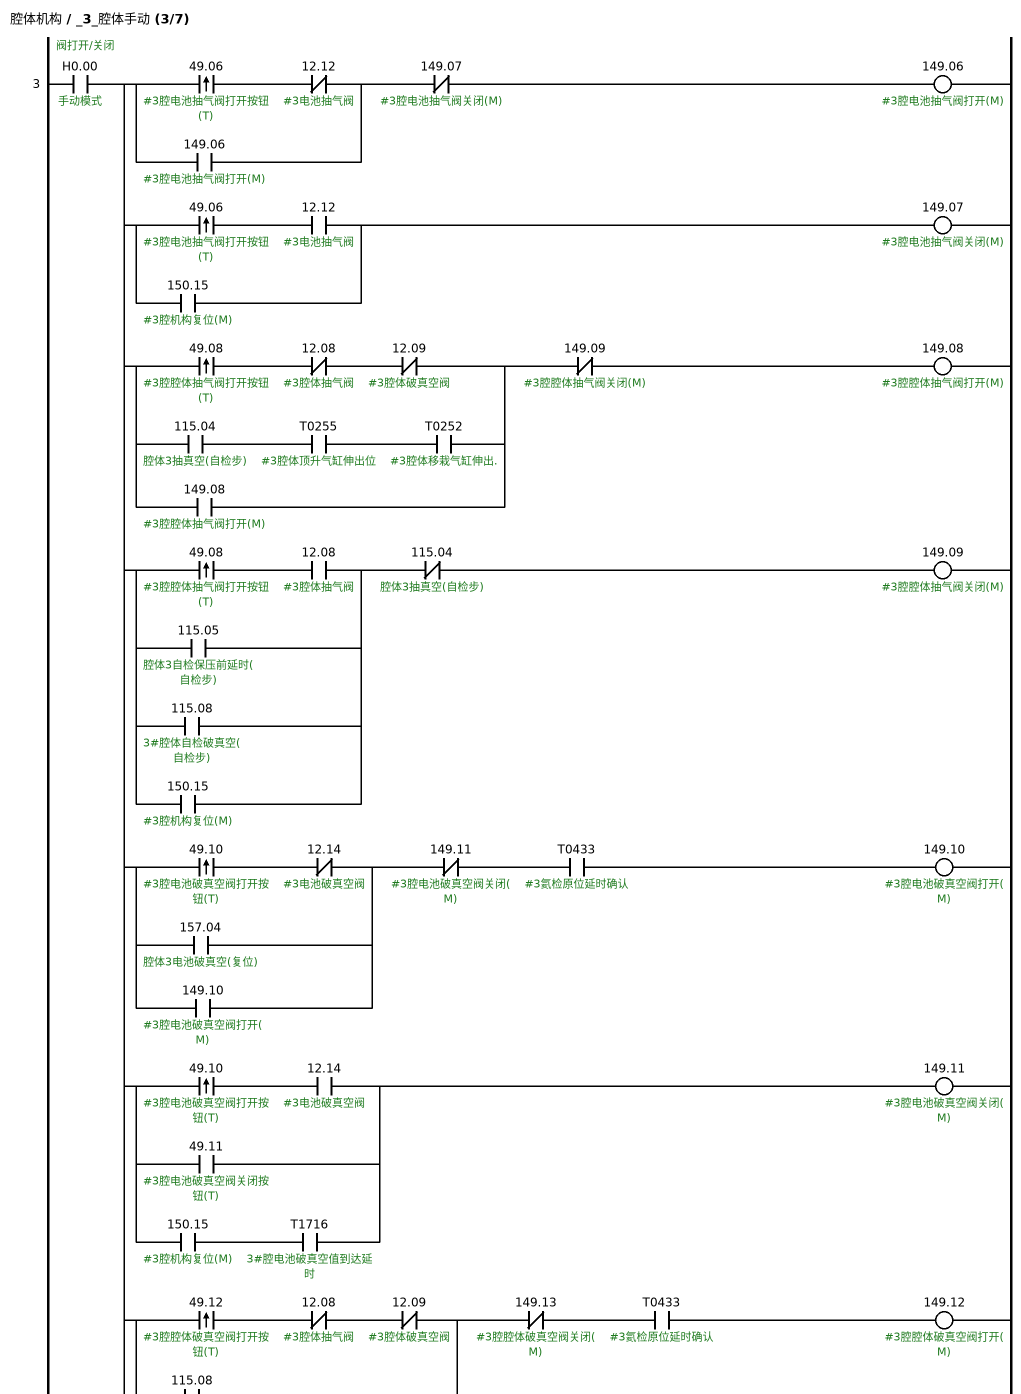
; [picture p264: 腔体机构 / _3_腔体手动, rungs 3-3]

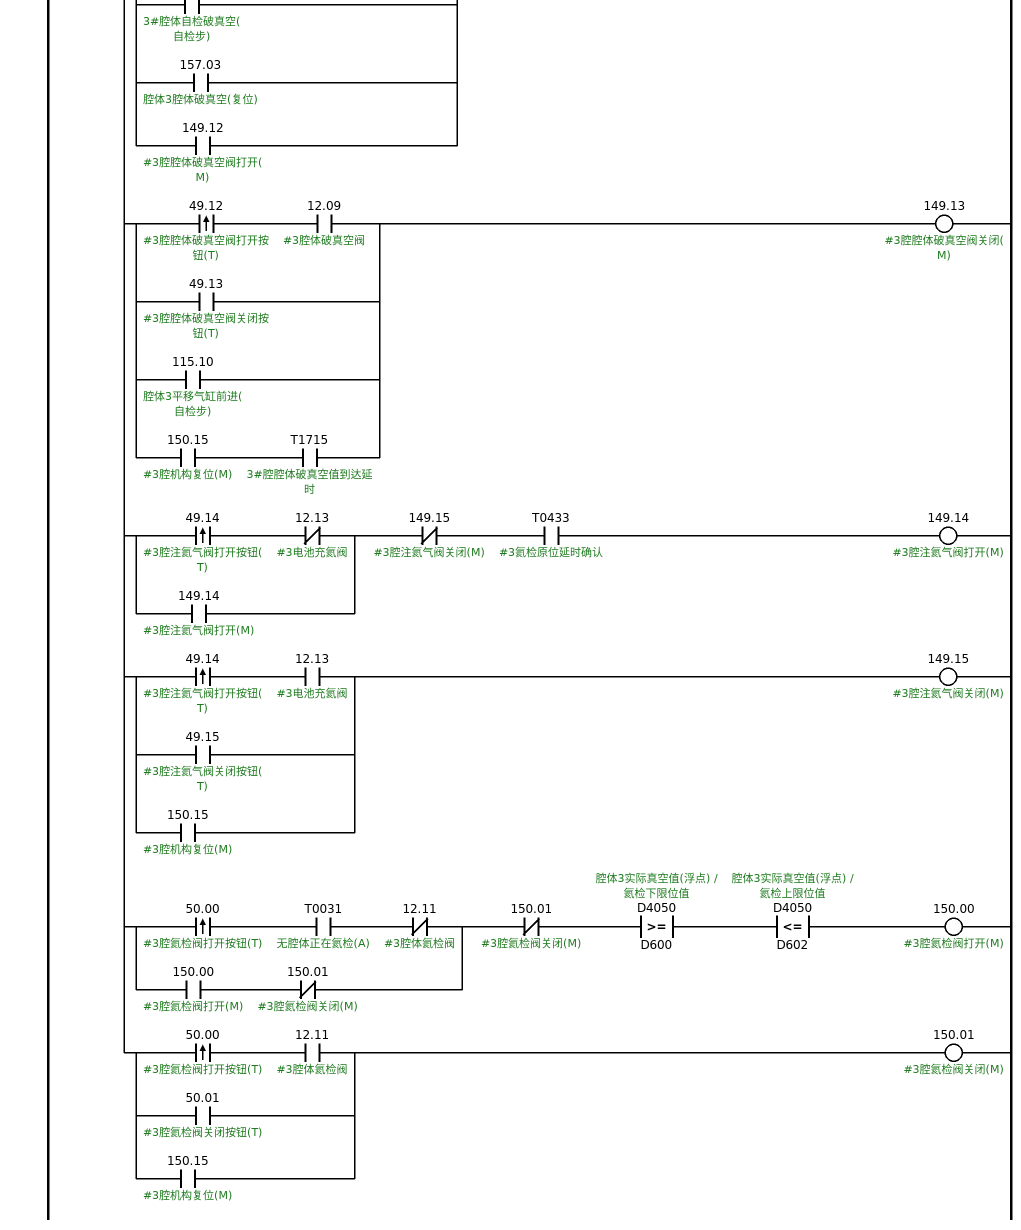
; rung 3: 阀打开/关闭
LD H0.00  ; 手动模式
OUT TR0
@LD 49.06  ; #3腔电池抽气阀打开按钮(T)
ANDNOT 12.12  ; #3电池抽气阀
OR 149.06  ; #3腔电池抽气阀打开(M)
ANDLD
ANDNOT 149.07  ; #3腔电池抽气阀关闭(M)
OUT 149.06  ; #3腔电池抽气阀打开(M)
LD TR0
@LD 49.06  ; #3腔电池抽气阀打开按钮(T)
AND 12.12  ; #3电池抽气阀
OR 150.15  ; #3腔机构复位(M)
ANDLD
OUT 149.07  ; #3腔电池抽气阀关闭(M)
LD TR0
@LD 49.08  ; #3腔腔体抽气阀打开按钮(T)
ANDNOT 12.08  ; #3腔体抽气阀
ANDNOT 12.09  ; #3腔体破真空阀
LD 115.04  ; 腔体3抽真空(自检步)
AND T0255  ; #3腔体顶升气缸伸出位
AND T0252  ; #3腔体移栽气缸伸出.
ORLD
OR 149.08  ; #3腔腔体抽气阀打开(M)
ANDLD
ANDNOT 149.09  ; #3腔腔体抽气阀关闭(M)
OUT 149.08  ; #3腔腔体抽气阀打开(M)
LD TR0
@LD 49.08  ; #3腔腔体抽气阀打开按钮(T)
AND 12.08  ; #3腔体抽气阀
OR 115.05  ; 腔体3自检保压前延时(自检步)
OR 115.08  ; 3#腔体自检破真空(自检步)
OR 150.15  ; #3腔机构复位(M)
ANDLD
ANDNOT 115.04  ; 腔体3抽真空(自检步)
OUT 149.09  ; #3腔腔体抽气阀关闭(M)
LD TR0
@LD 49.10  ; #3腔电池破真空阀打开按钮(T)
ANDNOT 12.14  ; #3电池破真空阀
OR 157.04  ; 腔体3电池破真空(复位)
OR 149.10  ; #3腔电池破真空阀打开(M)
ANDLD
ANDNOT 149.11  ; #3腔电池破真空阀关闭(M)
AND T0433  ; #3氦检原位延时确认
OUT 149.10  ; #3腔电池破真空阀打开(M)
LD TR0
@LD 49.10  ; #3腔电池破真空阀打开按钮(T)
AND 12.14  ; #3电池破真空阀
OR 49.11  ; #3腔电池破真空阀关闭按钮(T)
LD 150.15  ; #3腔机构复位(M)
AND T1716  ; 3#腔电池破真空值到达延时
ORLD
ANDLD
OUT 149.11  ; #3腔电池破真空阀关闭(M)
LD TR0
@LD 49.12  ; #3腔腔体破真空阀打开按钮(T)
ANDNOT 12.08  ; #3腔体抽气阀
ANDNOT 12.09  ; #3腔体破真空阀
OR 115.08  ; 3#腔体自检破真空(自检步)
OR 157.03  ; 腔体3腔体破真空(复位)
OR 149.12  ; #3腔腔体破真空阀打开(M)
ANDLD
ANDNOT 149.13  ; #3腔腔体破真空阀关闭(M)
AND T0433  ; #3氦检原位延时确认
OUT 149.12  ; #3腔腔体破真空阀打开(M)
LD TR0
@LD 49.12  ; #3腔腔体破真空阀打开按钮(T)
AND 12.09  ; #3腔体破真空阀
OR 49.13  ; #3腔腔体破真空阀关闭按钮(T)
OR 115.10  ; 腔体3平移气缸前进(自检步)
LD 150.15  ; #3腔机构复位(M)
AND T1715  ; 3#腔腔体破真空值到达延时
ORLD
ANDLD
OUT 149.13  ; #3腔腔体破真空阀关闭(M)
LD TR0
@LD 49.14  ; #3腔注氦气阀打开按钮(T)
ANDNOT 12.13  ; #3电池充氦阀
OR 149.14  ; #3腔注氦气阀打开(M)
ANDLD
ANDNOT 149.15  ; #3腔注氦气阀关闭(M)
AND T0433  ; #3氦检原位延时确认
OUT 149.14  ; #3腔注氦气阀打开(M)
LD TR0
@LD 49.14  ; #3腔注氦气阀打开按钮(T)
AND 12.13  ; #3电池充氦阀
OR 49.15  ; #3腔注氦气阀关闭按钮(T)
OR 150.15  ; #3腔机构复位(M)
ANDLD
OUT 149.15  ; #3腔注氦气阀关闭(M)
LD TR0
@LD 50.00  ; #3腔氦检阀打开按钮(T)
AND T0031  ; 无腔体正在氦检(A)
ANDNOT 12.11  ; #3腔体氦检阀
LD 150.00  ; #3腔氦检阀打开(M)
ANDNOT 150.01  ; #3腔氦检阀关闭(M)
ORLD
ANDLD
ANDNOT 150.01  ; #3腔氦检阀关闭(M)
AND>=F(334) D4050 D600  ; 腔体3实际真空值(浮点), 氦检下限位值
AND<=F(332) D4050 D602  ; 腔体3实际真空值(浮点), 氦检上限位值
OUT 150.00  ; #3腔氦检阀打开(M)
LD TR0
@LD 50.00  ; #3腔氦检阀打开按钮(T)
AND 12.11  ; #3腔体氦检阀
OR 50.01  ; #3腔氦检阀关闭按钮(T)
OR 150.15  ; #3腔机构复位(M)
ANDLD
OUT 150.01  ; #3腔氦检阀关闭(M)

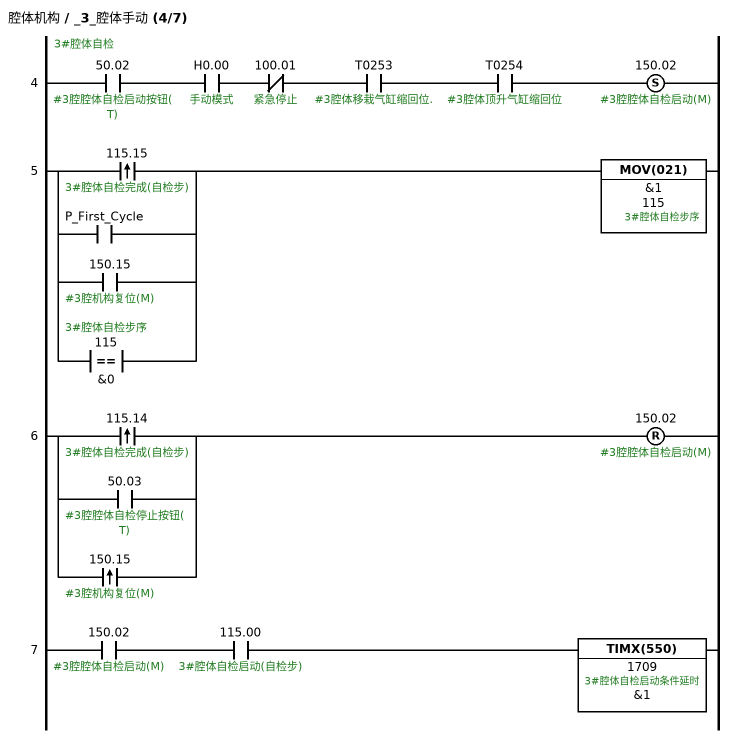
; rung 4: 3#腔体自检
LD 50.02  ; #3腔腔体自检启动按钮(T)
AND H0.00  ; 手动模式
ANDNOT 100.01  ; 紧急停止
AND T0253  ; #3腔体移栽气缸缩回位.
AND T0254  ; #3腔体顶升气缸缩回位
SET 150.02  ; #3腔腔体自检启动(M)
; rung 5
@LD 115.15  ; 3#腔体自检完成(自检步)
OR P_First_Cycle
OR 150.15  ; #3腔机构复位(M)
OR=(300) 115 &0  ; 3#腔体自检步序
MOV(021) &1 115  ; 3#腔体自检步序
; rung 6
@LD 115.14  ; 3#腔体自检完成(自检步)
OR 50.03  ; #3腔腔体自检停止按钮(T)
@OR 150.15  ; #3腔机构复位(M)
RSET 150.02  ; #3腔腔体自检启动(M)
; rung 7
LD 150.02  ; #3腔腔体自检启动(M)
AND 115.00  ; 3#腔体自检启动(自检步)
TIMX(550) 1709 &1  ; 3#腔体自检启动条件延时

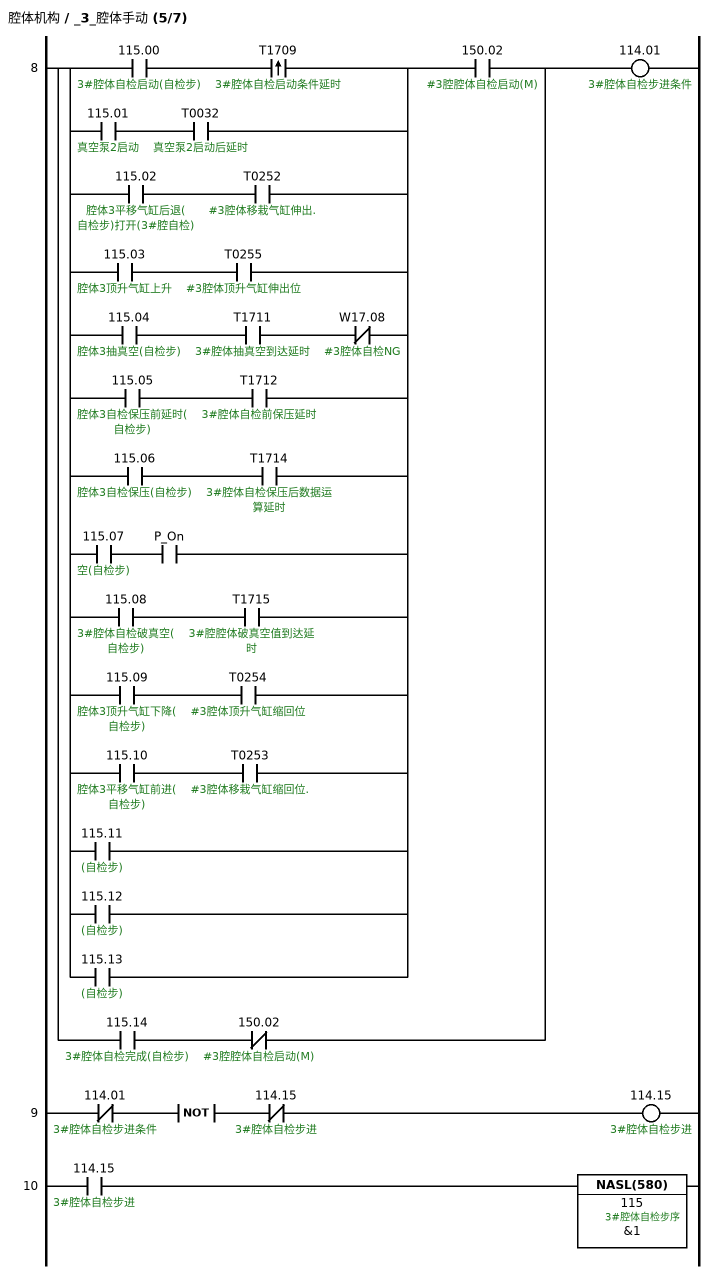
; rung 8
LD 115.00  ; 3#腔体自检启动(自检步)
@AND T1709  ; 3#腔体自检启动条件延时
LD 115.01  ; 真空泵2启动
AND T0032  ; 真空泵2启动后延时
ORLD
LD 115.02  ; 腔体3平移气缸后退(自检步)打开(3#腔自检)
AND T0252  ; #3腔体移栽气缸伸出.
ORLD
LD 115.03  ; 腔体3顶升气缸上升
AND T0255  ; #3腔体顶升气缸伸出位
ORLD
LD 115.04  ; 腔体3抽真空(自检步)
AND T1711  ; 3#腔体抽真空到达延时
ANDNOT W17.08  ; #3腔体自检NG
ORLD
LD 115.05  ; 腔体3自检保压前延时(自检步)
AND T1712  ; 3#腔体自检前保压延时
ORLD
LD 115.06  ; 腔体3自检保压(自检步)
AND T1714  ; 3#腔体自检保压后数据运算延时
ORLD
LD 115.07  ; 空(自检步)
AND P_On
ORLD
LD 115.08  ; 3#腔体自检破真空(自检步)
AND T1715  ; 3#腔腔体破真空值到达延时
ORLD
LD 115.09  ; 腔体3顶升气缸下降(自检步)
AND T0254  ; #3腔体顶升气缸缩回位
ORLD
LD 115.10  ; 腔体3平移气缸前进(自检步)
AND T0253  ; #3腔体移栽气缸缩回位.
ORLD
OR 115.11  ; (自检步)
OR 115.12  ; (自检步)
OR 115.13  ; (自检步)
AND 150.02  ; #3腔腔体自检启动(M)
LD 115.14  ; 3#腔体自检完成(自检步)
ANDNOT 150.02  ; #3腔腔体自检启动(M)
ORLD
OUT 114.01  ; 3#腔体自检步进条件
; rung 9
LDNOT 114.01  ; 3#腔体自检步进条件
NOT(520)
ANDNOT 114.15  ; 3#腔体自检步进
OUT 114.15  ; 3#腔体自检步进
; rung 10
LD 114.15  ; 3#腔体自检步进
NASL(580) 115 &1  ; 3#腔体自检步序

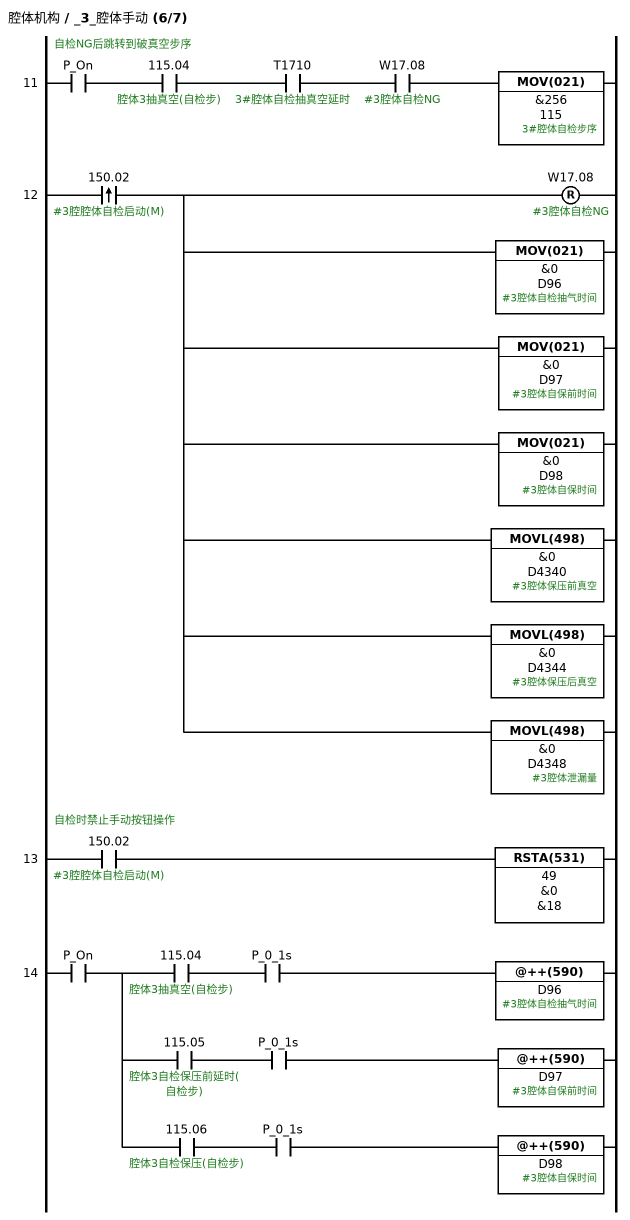
; rung 11: 自检NG后跳转到破真空步序
LD P_On
AND 115.04  ; 腔体3抽真空(自检步)
AND T1710  ; 3#腔体自检抽真空延时
AND W17.08  ; #3腔体自检NG
MOV(021) &256 115  ; 3#腔体自检步序
; rung 12
@LD 150.02  ; #3腔腔体自检启动(M)
RSET W17.08  ; #3腔体自检NG
MOV(021) &0 D96  ; #3腔体自检抽气时间
MOV(021) &0 D97  ; #3腔体自保前时间
MOV(021) &0 D98  ; #3腔体自保时间
MOVL(498) &0 D4340  ; #3腔体保压前真空
MOVL(498) &0 D4344  ; #3腔体保压后真空
MOVL(498) &0 D4348  ; #3腔体泄漏量
; rung 13: 自检时禁止手动按钮操作
LD 150.02  ; #3腔腔体自检启动(M)
RSTA(531) 49 &0 &18
; rung 14
LD P_On
OUT TR0
AND 115.04  ; 腔体3抽真空(自检步)
AND P_0_1s
@++(590) D96  ; #3腔体自检抽气时间
LD TR0
AND 115.05  ; 腔体3自检保压前延时(自检步)
AND P_0_1s
@++(590) D97  ; #3腔体自保前时间
LD TR0
AND 115.06  ; 腔体3自检保压(自检步)
AND P_0_1s
@++(590) D98  ; #3腔体自保时间

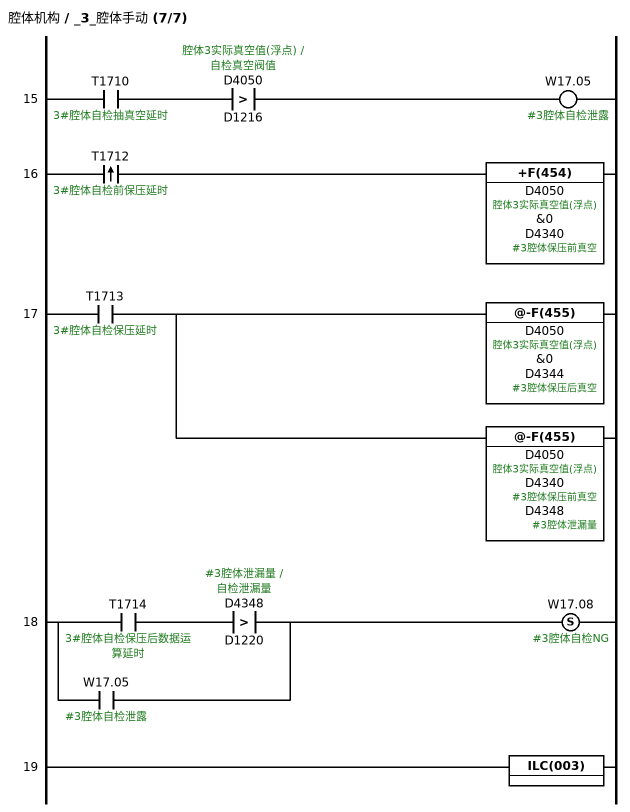
; rung 15
LD T1710  ; 3#腔体自检抽真空延时
AND>F(333) D4050 D1216  ; 腔体3实际真空值(浮点), 自检真空阀值
OUT W17.05  ; #3腔体自检泄露
; rung 16
@LD T1712  ; 3#腔体自检前保压延时
+F(454) D4050 &0 D4340  ; 腔体3实际真空值(浮点), #3腔体保压前真空
; rung 17
LD T1713  ; 3#腔体自检保压延时
@-F(455) D4050 &0 D4344  ; 腔体3实际真空值(浮点), #3腔体保压后真空
@-F(455) D4050 D4340 D4348  ; 腔体3实际真空值(浮点), #3腔体保压前真空, #3腔体泄漏量
; rung 18
LD T1714  ; 3#腔体自检保压后数据运算延时
AND>F(333) D4348 D1220  ; #3腔体泄漏量, 自检泄漏量
OR W17.05  ; #3腔体自检泄露
SET W17.08  ; #3腔体自检NG
; rung 19
ILC(003)

### Section _4_腔体手动

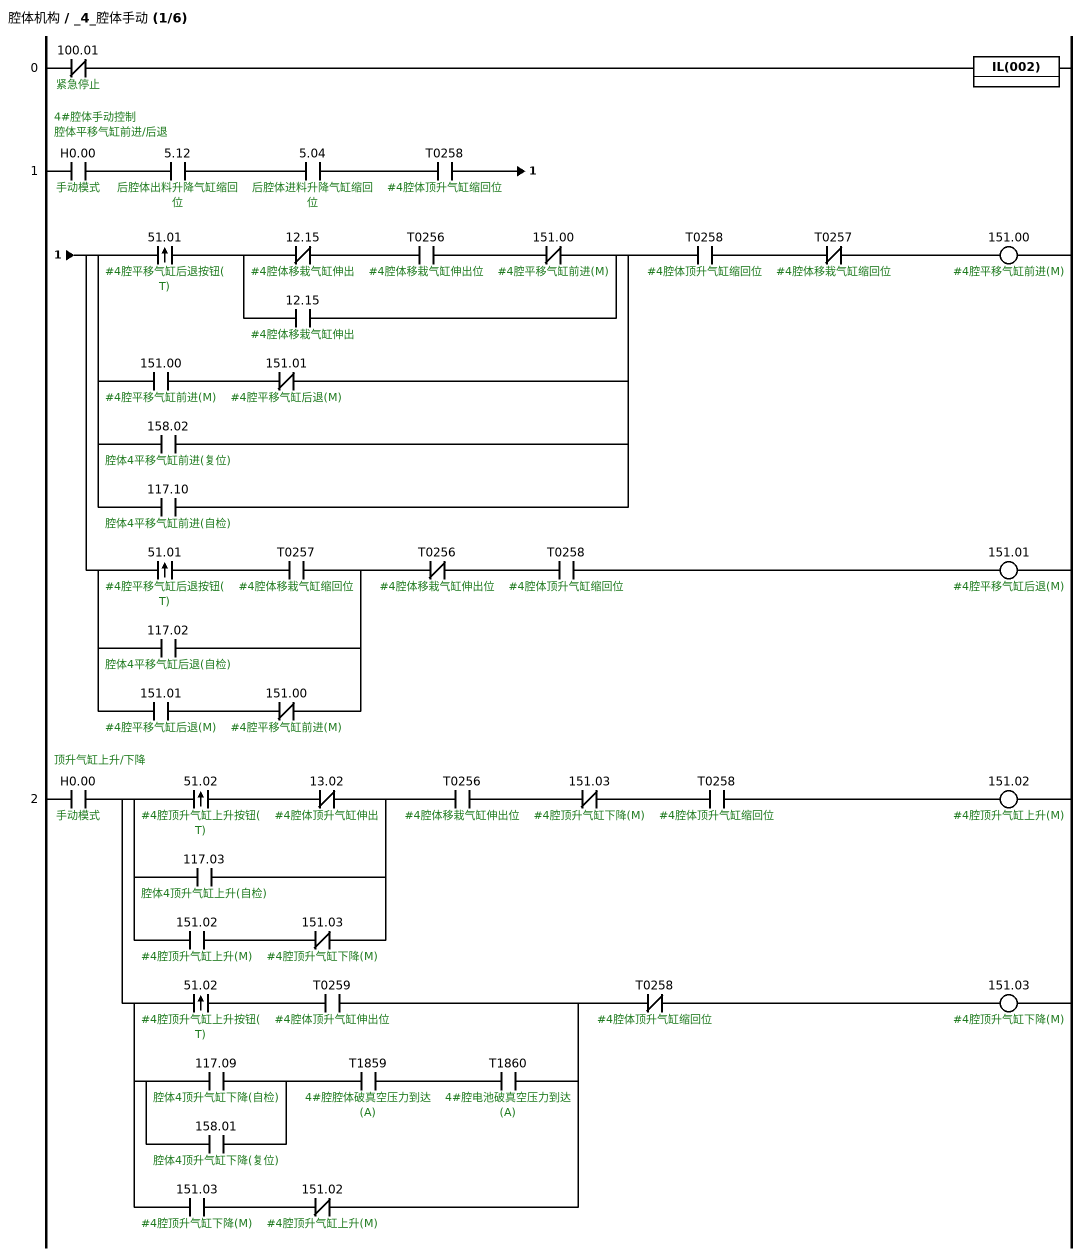
; rung 0
LDNOT 100.01  ; 紧急停止
IL(002)
; rung 1: 4#腔体手动控制 / 腔体平移气缸前进/后退
LD H0.00  ; 手动模式
AND 5.12  ; 后腔体出料升降气缸缩回位
AND 5.04  ; 后腔体进料升降气缸缩回位
AND T0258  ; #4腔体顶升气缸缩回位
OUT TR0
@LD 51.01  ; #4腔平移气缸后退按钮(T)
LDNOT 12.15  ; #4腔体移栽气缸伸出
AND T0256  ; #4腔体移栽气缸伸出位
ANDNOT 151.00  ; #4腔平移气缸前进(M)
OR 12.15  ; #4腔体移栽气缸伸出
ANDLD
LD 151.00  ; #4腔平移气缸前进(M)
ANDNOT 151.01  ; #4腔平移气缸后退(M)
ORLD
OR 158.02  ; 腔体4平移气缸前进(复位)
OR 117.10  ; 腔体4平移气缸前进(自检)
ANDLD
AND T0258  ; #4腔体顶升气缸缩回位
ANDNOT T0257  ; #4腔体移栽气缸缩回位
OUT 151.00  ; #4腔平移气缸前进(M)
LD TR0
@LD 51.01  ; #4腔平移气缸后退按钮(T)
AND T0257  ; #4腔体移栽气缸缩回位
OR 117.02  ; 腔体4平移气缸后退(自检)
LD 151.01  ; #4腔平移气缸后退(M)
ANDNOT 151.00  ; #4腔平移气缸前进(M)
ORLD
ANDLD
ANDNOT T0256  ; #4腔体移栽气缸伸出位
AND T0258  ; #4腔体顶升气缸缩回位
OUT 151.01  ; #4腔平移气缸后退(M)
; rung 2: 顶升气缸上升/下降
LD H0.00  ; 手动模式
OUT TR0
@LD 51.02  ; #4腔顶升气缸上升按钮(T)
ANDNOT 13.02  ; #4腔体顶升气缸伸出
OR 117.03  ; 腔体4顶升气缸上升(自检)
LD 151.02  ; #4腔顶升气缸上升(M)
ANDNOT 151.03  ; #4腔顶升气缸下降(M)
ORLD
ANDLD
AND T0256  ; #4腔体移栽气缸伸出位
ANDNOT 151.03  ; #4腔顶升气缸下降(M)
AND T0258  ; #4腔体顶升气缸缩回位
OUT 151.02  ; #4腔顶升气缸上升(M)
LD TR0
@LD 51.02  ; #4腔顶升气缸上升按钮(T)
AND T0259  ; #4腔体顶升气缸伸出位
LD 117.09  ; 腔体4顶升气缸下降(自检)
OR 158.01  ; 腔体4顶升气缸下降(复位)
AND T1859  ; 4#腔腔体破真空压力到达(A)
AND T1860  ; 4#腔电池破真空压力到达(A)
ORLD
LD 151.03  ; #4腔顶升气缸下降(M)
ANDNOT 151.02  ; #4腔顶升气缸上升(M)
ORLD
ANDLD
ANDNOT T0258  ; #4腔体顶升气缸缩回位
OUT 151.03  ; #4腔顶升气缸下降(M)

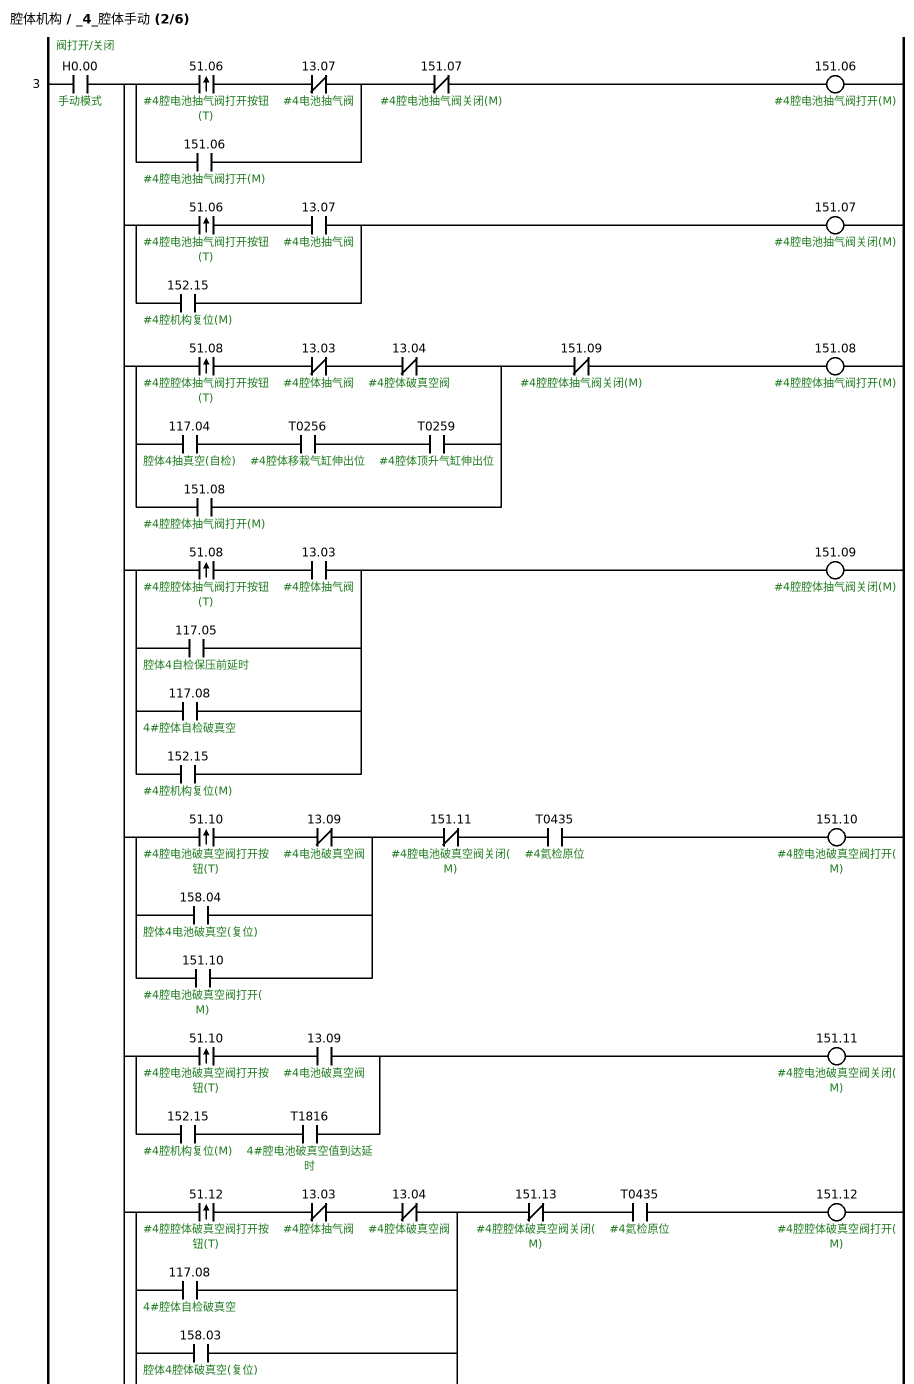

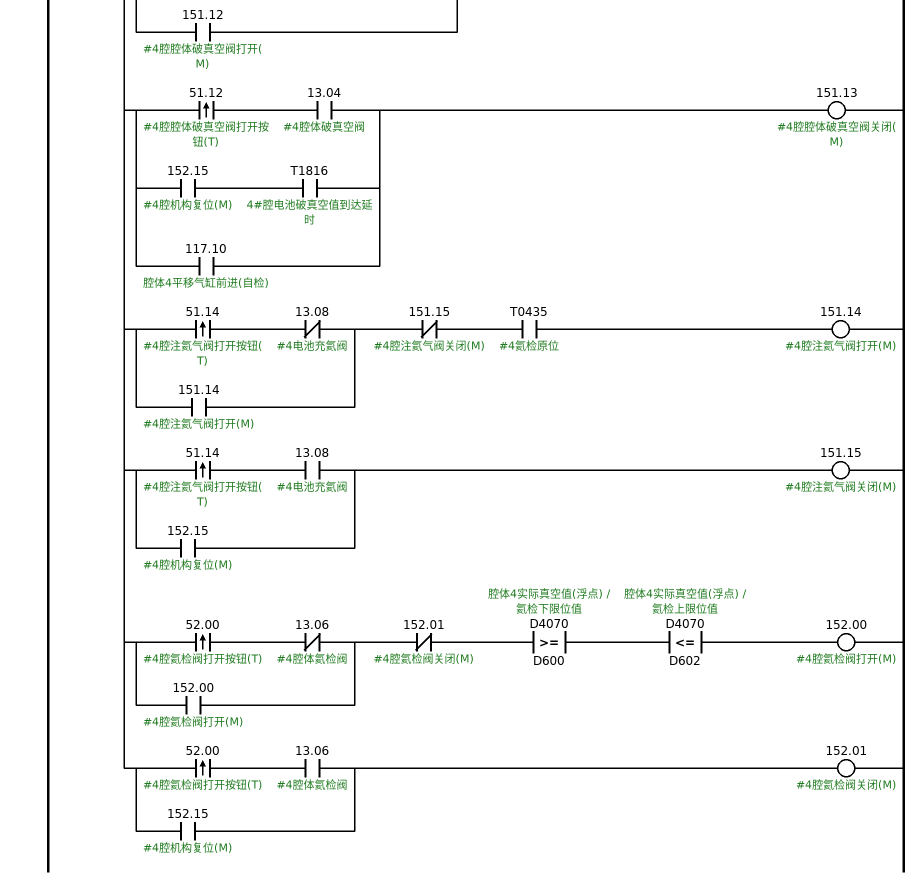
; rung 3: 阀打开/关闭
LD H0.00  ; 手动模式
OUT TR0
@LD 51.06  ; #4腔电池抽气阀打开按钮(T)
ANDNOT 13.07  ; #4电池抽气阀
OR 151.06  ; #4腔电池抽气阀打开(M)
ANDLD
ANDNOT 151.07  ; #4腔电池抽气阀关闭(M)
OUT 151.06  ; #4腔电池抽气阀打开(M)
LD TR0
@LD 51.06  ; #4腔电池抽气阀打开按钮(T)
AND 13.07  ; #4电池抽气阀
OR 152.15  ; #4腔机构复位(M)
ANDLD
OUT 151.07  ; #4腔电池抽气阀关闭(M)
LD TR0
@LD 51.08  ; #4腔腔体抽气阀打开按钮(T)
ANDNOT 13.03  ; #4腔体抽气阀
ANDNOT 13.04  ; #4腔体破真空阀
LD 117.04  ; 腔体4抽真空(自检)
AND T0256  ; #4腔体移栽气缸伸出位
AND T0259  ; #4腔体顶升气缸伸出位
ORLD
OR 151.08  ; #4腔腔体抽气阀打开(M)
ANDLD
ANDNOT 151.09  ; #4腔腔体抽气阀关闭(M)
OUT 151.08  ; #4腔腔体抽气阀打开(M)
LD TR0
@LD 51.08  ; #4腔腔体抽气阀打开按钮(T)
AND 13.03  ; #4腔体抽气阀
OR 117.05  ; 腔体4自检保压前延时
OR 117.08  ; 4#腔体自检破真空
OR 152.15  ; #4腔机构复位(M)
ANDLD
OUT 151.09  ; #4腔腔体抽气阀关闭(M)
LD TR0
@LD 51.10  ; #4腔电池破真空阀打开按钮(T)
ANDNOT 13.09  ; #4电池破真空阀
OR 158.04  ; 腔体4电池破真空(复位)
OR 151.10  ; #4腔电池破真空阀打开(M)
ANDLD
ANDNOT 151.11  ; #4腔电池破真空阀关闭(M)
AND T0435  ; #4氦检原位
OUT 151.10  ; #4腔电池破真空阀打开(M)
LD TR0
@LD 51.10  ; #4腔电池破真空阀打开按钮(T)
AND 13.09  ; #4电池破真空阀
LD 152.15  ; #4腔机构复位(M)
AND T1816  ; 4#腔电池破真空值到达延时
ORLD
ANDLD
OUT 151.11  ; #4腔电池破真空阀关闭(M)
LD TR0
@LD 51.12  ; #4腔腔体破真空阀打开按钮(T)
ANDNOT 13.03  ; #4腔体抽气阀
ANDNOT 13.04  ; #4腔体破真空阀
OR 117.08  ; 4#腔体自检破真空
OR 158.03  ; 腔体4腔体破真空(复位)
OR 151.12  ; #4腔腔体破真空阀打开(M)
ANDLD
ANDNOT 151.13  ; #4腔腔体破真空阀关闭(M)
AND T0435  ; #4氦检原位
OUT 151.12  ; #4腔腔体破真空阀打开(M)
LD TR0
@LD 51.12  ; #4腔腔体破真空阀打开按钮(T)
AND 13.04  ; #4腔体破真空阀
LD 152.15  ; #4腔机构复位(M)
AND T1816  ; 4#腔电池破真空值到达延时
ORLD
OR 117.10  ; 腔体4平移气缸前进(自检)
ANDLD
OUT 151.13  ; #4腔腔体破真空阀关闭(M)
LD TR0
@LD 51.14  ; #4腔注氦气阀打开按钮(T)
ANDNOT 13.08  ; #4电池充氦阀
OR 151.14  ; #4腔注氦气阀打开(M)
ANDLD
ANDNOT 151.15  ; #4腔注氦气阀关闭(M)
AND T0435  ; #4氦检原位
OUT 151.14  ; #4腔注氦气阀打开(M)
LD TR0
@LD 51.14  ; #4腔注氦气阀打开按钮(T)
AND 13.08  ; #4电池充氦阀
OR 152.15  ; #4腔机构复位(M)
ANDLD
OUT 151.15  ; #4腔注氦气阀关闭(M)
LD TR0
@LD 52.00  ; #4腔氦检阀打开按钮(T)
ANDNOT 13.06  ; #4腔体氦检阀
OR 152.00  ; #4腔氦检阀打开(M)
ANDLD
ANDNOT 152.01  ; #4腔氦检阀关闭(M)
AND>=F(334) D4070 D600  ; 腔体4实际真空值(浮点), 氦检下限位值
AND<=F(332) D4070 D602  ; 腔体4实际真空值(浮点), 氦检上限位值
OUT 152.00  ; #4腔氦检阀打开(M)
LD TR0
@LD 52.00  ; #4腔氦检阀打开按钮(T)
AND 13.06  ; #4腔体氦检阀
OR 152.15  ; #4腔机构复位(M)
ANDLD
OUT 152.01  ; #4腔氦检阀关闭(M)

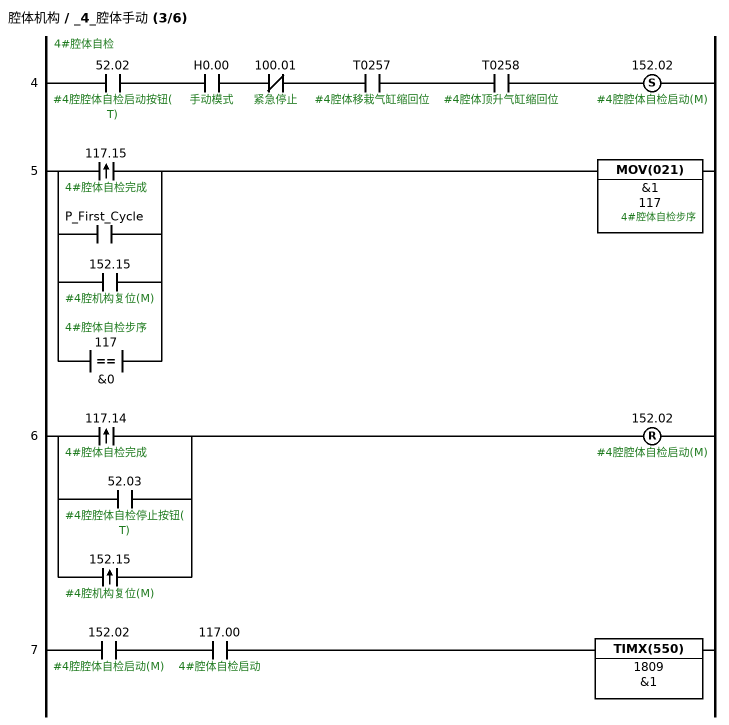
; rung 4: 4#腔体自检
LD 52.02  ; #4腔腔体自检启动按钮(T)
AND H0.00  ; 手动模式
ANDNOT 100.01  ; 紧急停止
AND T0257  ; #4腔体移栽气缸缩回位
AND T0258  ; #4腔体顶升气缸缩回位
SET 152.02  ; #4腔腔体自检启动(M)
; rung 5
@LD 117.15  ; 4#腔体自检完成
OR P_First_Cycle
OR 152.15  ; #4腔机构复位(M)
OR=(300) 117 &0  ; 4#腔体自检步序
MOV(021) &1 117  ; 4#腔体自检步序
; rung 6
@LD 117.14  ; 4#腔体自检完成
OR 52.03  ; #4腔腔体自检停止按钮(T)
@OR 152.15  ; #4腔机构复位(M)
RSET 152.02  ; #4腔腔体自检启动(M)
; rung 7
LD 152.02  ; #4腔腔体自检启动(M)
AND 117.00  ; 4#腔体自检启动
TIMX(550) 1809 &1

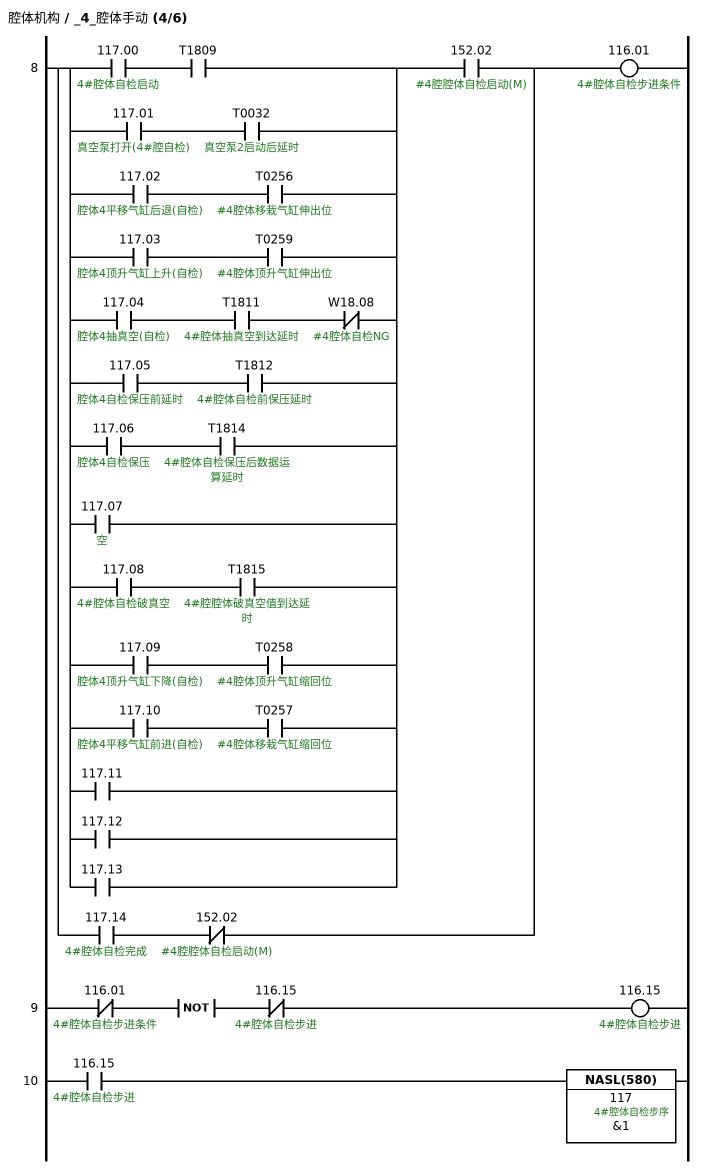
; rung 8
LD 117.00  ; 4#腔体自检启动
AND T1809
LD 117.01  ; 真空泵打开(4#腔自检)
AND T0032  ; 真空泵2启动后延时
ORLD
LD 117.02  ; 腔体4平移气缸后退(自检)
AND T0256  ; #4腔体移栽气缸伸出位
ORLD
LD 117.03  ; 腔体4顶升气缸上升(自检)
AND T0259  ; #4腔体顶升气缸伸出位
ORLD
LD 117.04  ; 腔体4抽真空(自检)
AND T1811  ; 4#腔体抽真空到达延时
ANDNOT W18.08  ; #4腔体自检NG
ORLD
LD 117.05  ; 腔体4自检保压前延时
AND T1812  ; 4#腔体自检前保压延时
ORLD
LD 117.06  ; 腔体4自检保压
AND T1814  ; 4#腔体自检保压后数据运算延时
ORLD
OR 117.07  ; 空
LD 117.08  ; 4#腔体自检破真空
AND T1815  ; 4#腔腔体破真空值到达延时
ORLD
LD 117.09  ; 腔体4顶升气缸下降(自检)
AND T0258  ; #4腔体顶升气缸缩回位
ORLD
LD 117.10  ; 腔体4平移气缸前进(自检)
AND T0257  ; #4腔体移栽气缸缩回位
ORLD
OR 117.11
OR 117.12
OR 117.13
AND 152.02  ; #4腔腔体自检启动(M)
LD 117.14  ; 4#腔体自检完成
ANDNOT 152.02  ; #4腔腔体自检启动(M)
ORLD
OUT 116.01  ; 4#腔体自检步进条件
; rung 9
LDNOT 116.01  ; 4#腔体自检步进条件
NOT(520)
ANDNOT 116.15  ; 4#腔体自检步进
OUT 116.15  ; 4#腔体自检步进
; rung 10
LD 116.15  ; 4#腔体自检步进
NASL(580) 117 &1  ; 4#腔体自检步序

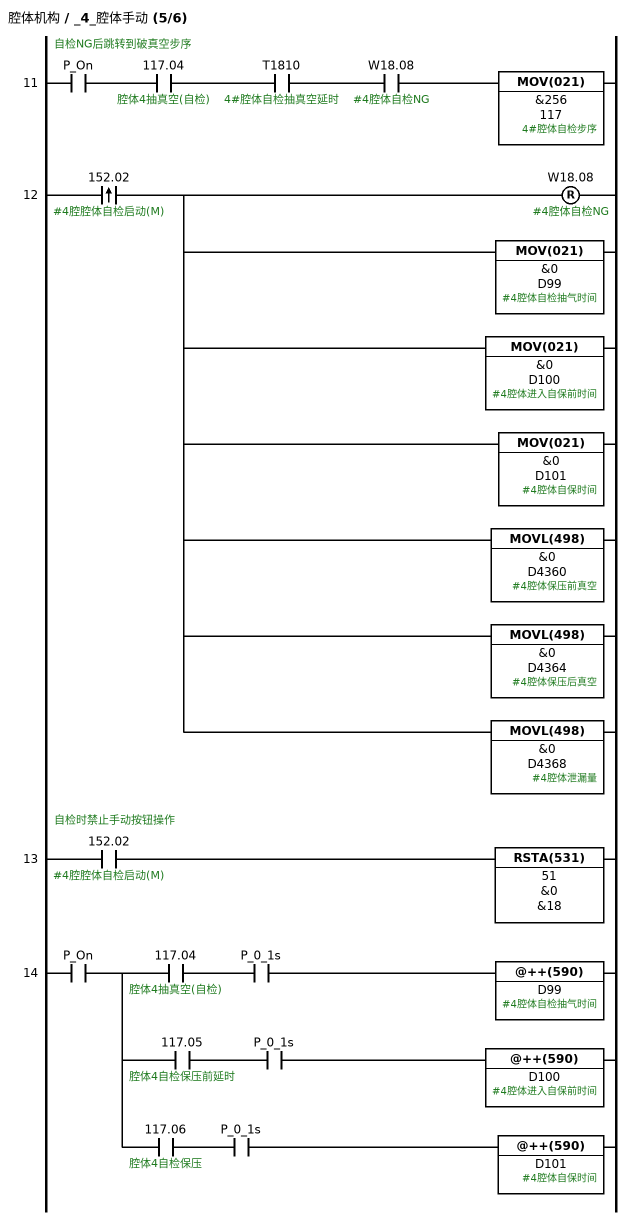
; rung 11: 自检NG后跳转到破真空步序
LD P_On
AND 117.04  ; 腔体4抽真空(自检)
AND T1810  ; 4#腔体自检抽真空延时
AND W18.08  ; #4腔体自检NG
MOV(021) &256 117  ; 4#腔体自检步序
; rung 12
@LD 152.02  ; #4腔腔体自检启动(M)
RSET W18.08  ; #4腔体自检NG
MOV(021) &0 D99  ; #4腔体自检抽气时间
MOV(021) &0 D100  ; #4腔体进入自保前时间
MOV(021) &0 D101  ; #4腔体自保时间
MOVL(498) &0 D4360  ; #4腔体保压前真空
MOVL(498) &0 D4364  ; #4腔体保压后真空
MOVL(498) &0 D4368  ; #4腔体泄漏量
; rung 13: 自检时禁止手动按钮操作
LD 152.02  ; #4腔腔体自检启动(M)
RSTA(531) 51 &0 &18
; rung 14
LD P_On
OUT TR0
AND 117.04  ; 腔体4抽真空(自检)
AND P_0_1s
@++(590) D99  ; #4腔体自检抽气时间
LD TR0
AND 117.05  ; 腔体4自检保压前延时
AND P_0_1s
@++(590) D100  ; #4腔体进入自保前时间
LD TR0
AND 117.06  ; 腔体4自检保压
AND P_0_1s
@++(590) D101  ; #4腔体自保时间

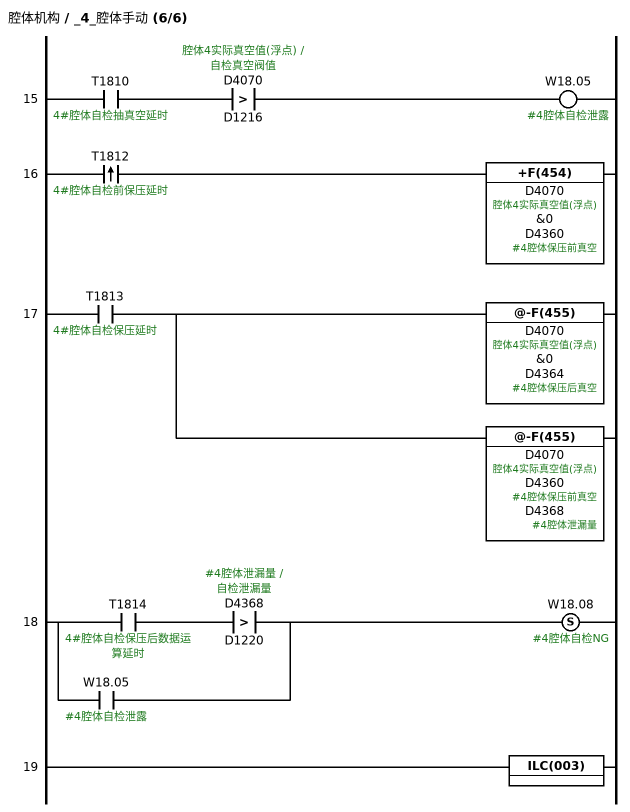
; rung 15
LD T1810  ; 4#腔体自检抽真空延时
AND>F(333) D4070 D1216  ; 腔体4实际真空值(浮点), 自检真空阀值
OUT W18.05  ; #4腔体自检泄露
; rung 16
@LD T1812  ; 4#腔体自检前保压延时
+F(454) D4070 &0 D4360  ; 腔体4实际真空值(浮点), #4腔体保压前真空
; rung 17
LD T1813  ; 4#腔体自检保压延时
@-F(455) D4070 &0 D4364  ; 腔体4实际真空值(浮点), #4腔体保压后真空
@-F(455) D4070 D4360 D4368  ; 腔体4实际真空值(浮点), #4腔体保压前真空, #4腔体泄漏量
; rung 18
LD T1814  ; 4#腔体自检保压后数据运算延时
AND>F(333) D4368 D1220  ; #4腔体泄漏量, 自检泄漏量
OR W18.05  ; #4腔体自检泄露
SET W18.08  ; #4腔体自检NG
; rung 19
ILC(003)

### Section _1_腔体自动

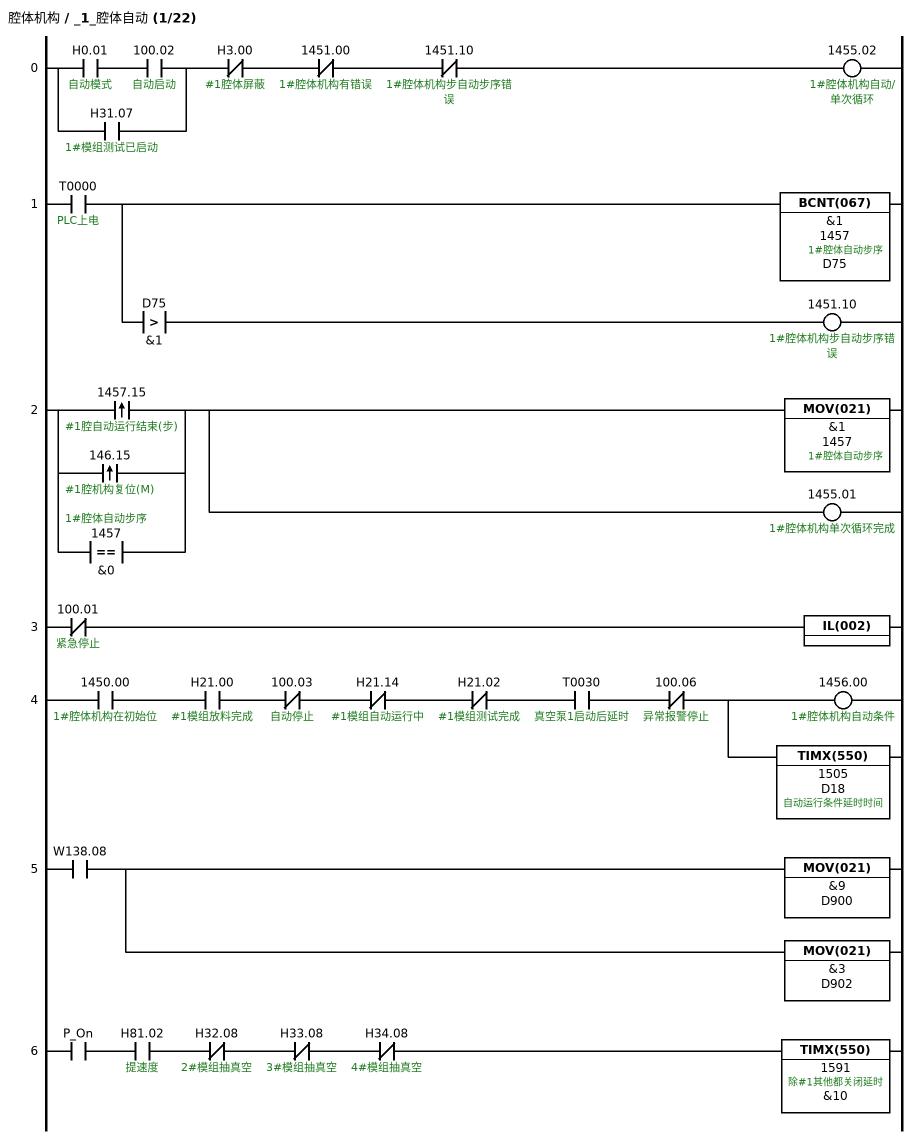
; rung 0
LD H0.01  ; 自动模式
AND 100.02  ; 自动启动
OR H31.07  ; 1#模组测试已启动
ANDNOT H3.00  ; #1腔体屏蔽
ANDNOT 1451.00  ; 1#腔体机构有错误
ANDNOT 1451.10  ; 1#腔体机构步自动步序错误
OUT 1455.02  ; 1#腔体机构自动/单次循环
; rung 1
LD T0000  ; PLC上电
BCNT(067) &1 1457 D75  ; 1#腔体自动步序
AND>(320) D75 &1
OUT 1451.10  ; 1#腔体机构步自动步序错误
; rung 2
@LD 1457.15  ; #1腔自动运行结束(步)
@OR 146.15  ; #1腔机构复位(M)
OR=(300) 1457 &0  ; 1#腔体自动步序
MOV(021) &1 1457  ; 1#腔体自动步序
OUT 1455.01  ; 1#腔体机构单次循环完成
; rung 3
LDNOT 100.01  ; 紧急停止
IL(002)
; rung 4
LD 1450.00  ; 1#腔体机构在初始位
AND H21.00  ; #1模组放料完成
ANDNOT 100.03  ; 自动停止
ANDNOT H21.14  ; #1模组自动运行中
ANDNOT H21.02  ; #1模组测试完成
AND T0030  ; 真空泵1启动后延时
ANDNOT 100.06  ; 异常报警停止
OUT 1456.00  ; 1#腔体机构自动条件
TIMX(550) 1505 D18  ; 自动运行条件延时时间
; rung 5
LD W138.08
MOV(021) &9 D900
MOV(021) &3 D902
; rung 6
LD P_On
AND H81.02  ; 提速度
ANDNOT H32.08  ; 2#模组抽真空
ANDNOT H33.08  ; 3#模组抽真空
ANDNOT H34.08  ; 4#模组抽真空
TIMX(550) 1591 &10  ; 除#1其他都关闭延时

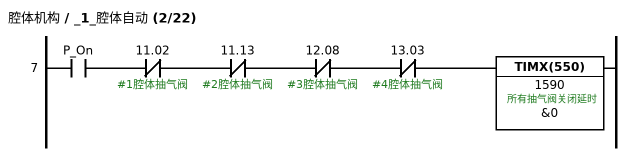
; rung 7
LD P_On
ANDNOT 11.02  ; #1腔体抽气阀
ANDNOT 11.13  ; #2腔体抽气阀
ANDNOT 12.08  ; #3腔体抽气阀
ANDNOT 13.03  ; #4腔体抽气阀
TIMX(550) 1590 &0  ; 所有抽气阀关闭延时

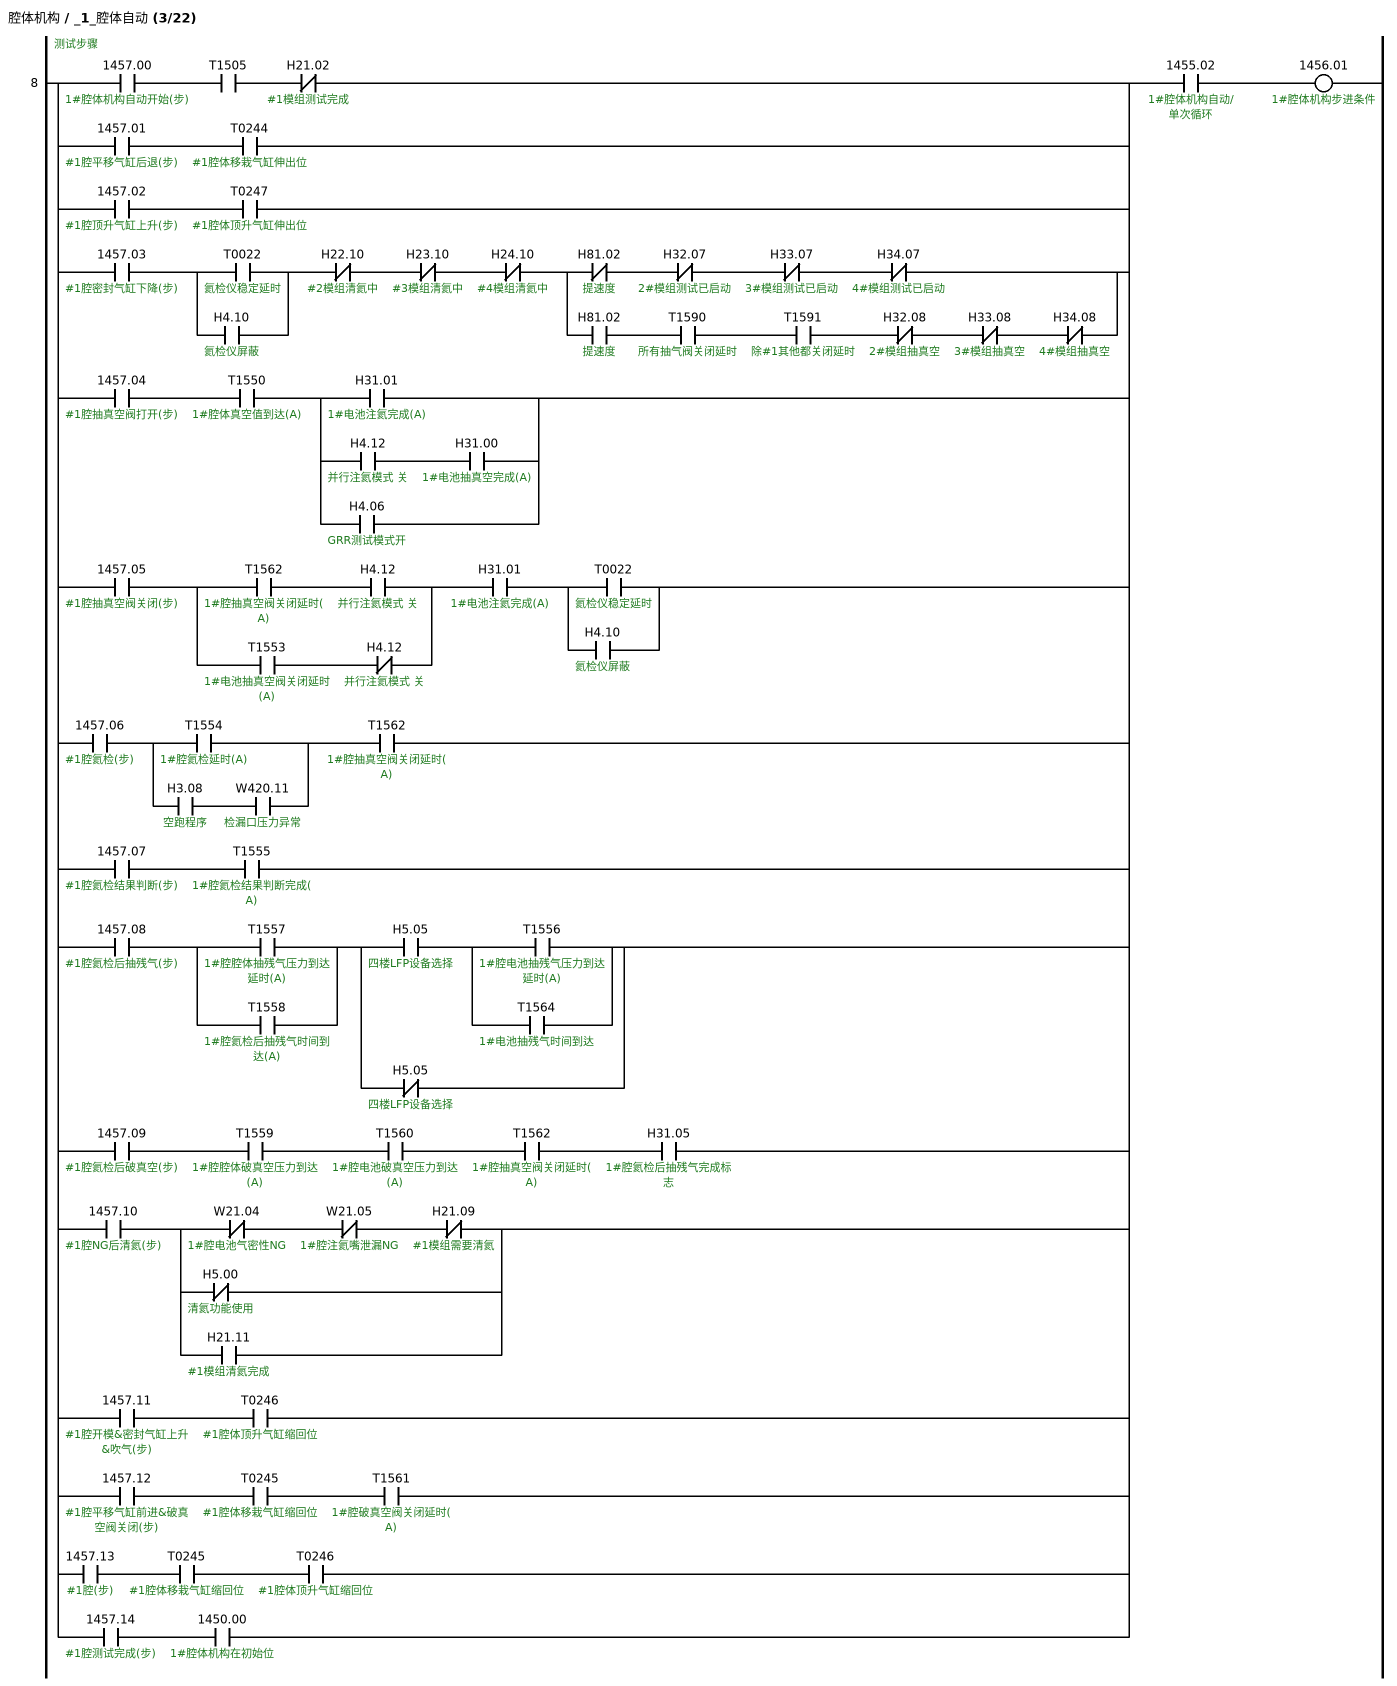
; rung 8: 测试步骤
LD 1457.00  ; 1#腔体机构自动开始(步)
AND T1505
ANDNOT H21.02  ; #1模组测试完成
LD 1457.01  ; #1腔平移气缸后退(步)
AND T0244  ; #1腔体移栽气缸伸出位
ORLD
LD 1457.02  ; #1腔顶升气缸上升(步)
AND T0247  ; #1腔体顶升气缸伸出位
ORLD
LD 1457.03  ; #1腔密封气缸下降(步)
LD T0022  ; 氦检仪稳定延时
OR H4.10  ; 氦检仪屏蔽
ANDLD
ANDNOT H22.10  ; #2模组清氦中
ANDNOT H23.10  ; #3模组清氦中
ANDNOT H24.10  ; #4模组清氦中
LDNOT H81.02  ; 提速度
ANDNOT H32.07  ; 2#模组测试已启动
ANDNOT H33.07  ; 3#模组测试已启动
ANDNOT H34.07  ; 4#模组测试已启动
LD H81.02  ; 提速度
AND T1590  ; 所有抽气阀关闭延时
AND T1591  ; 除#1其他都关闭延时
ANDNOT H32.08  ; 2#模组抽真空
ANDNOT H33.08  ; 3#模组抽真空
ANDNOT H34.08  ; 4#模组抽真空
ORLD
ANDLD
ORLD
LD 1457.04  ; #1腔抽真空阀打开(步)
AND T1550  ; 1#腔体真空值到达(A)
LD H31.01  ; 1#电池注氦完成(A)
LD H4.12  ; 并行注氦模式 关
AND H31.00  ; 1#电池抽真空完成(A)
ORLD
OR H4.06  ; GRR测试模式开
ANDLD
ORLD
LD 1457.05  ; #1腔抽真空阀关闭(步)
LD T1562  ; 1#腔抽真空阀关闭延时(A)
AND H4.12  ; 并行注氦模式 关
LD T1553  ; 1#电池抽真空阀关闭延时(A)
ANDNOT H4.12  ; 并行注氦模式 关
ORLD
ANDLD
AND H31.01  ; 1#电池注氦完成(A)
LD T0022  ; 氦检仪稳定延时
OR H4.10  ; 氦检仪屏蔽
ANDLD
ORLD
LD 1457.06  ; #1腔氦检(步)
LD T1554  ; 1#腔氦检延时(A)
LD H3.08  ; 空跑程序
AND W420.11  ; 检漏口压力异常
ORLD
ANDLD
AND T1562  ; 1#腔抽真空阀关闭延时(A)
ORLD
LD 1457.07  ; #1腔氦检结果判断(步)
AND T1555  ; 1#腔氦检结果判断完成(A)
ORLD
LD 1457.08  ; #1腔氦检后抽残气(步)
LD T1557  ; 1#腔腔体抽残气压力到达延时(A)
OR T1558  ; 1#腔氦检后抽残气时间到达(A)
ANDLD
LD H5.05  ; 四楼LFP设备选择
LD T1556  ; 1#腔电池抽残气压力到达延时(A)
OR T1564  ; 1#电池抽残气时间到达
ANDLD
ORNOT H5.05  ; 四楼LFP设备选择
ANDLD
ORLD
LD 1457.09  ; #1腔氦检后破真空(步)
AND T1559  ; 1#腔腔体破真空压力到达(A)
AND T1560  ; 1#腔电池破真空压力到达(A)
AND T1562  ; 1#腔抽真空阀关闭延时(A)
AND H31.05  ; 1#腔氦检后抽残气完成标志
ORLD
LD 1457.10  ; #1腔NG后清氦(步)
LDNOT W21.04  ; 1#腔电池气密性NG
ANDNOT W21.05  ; 1#腔注氦嘴泄漏NG
ANDNOT H21.09  ; #1模组需要清氦
ORNOT H5.00  ; 清氦功能使用
OR H21.11  ; #1模组清氦完成
ANDLD
ORLD
LD 1457.11  ; #1腔开模&密封气缸上升&吹气(步)
AND T0246  ; #1腔体顶升气缸缩回位
ORLD
LD 1457.12  ; #1腔平移气缸前进&破真空阀关闭(步)
AND T0245  ; #1腔体移栽气缸缩回位
AND T1561  ; 1#腔破真空阀关闭延时(A)
ORLD
LD 1457.13  ; #1腔(步)
AND T0245  ; #1腔体移栽气缸缩回位
AND T0246  ; #1腔体顶升气缸缩回位
ORLD
LD 1457.14  ; #1腔测试完成(步)
AND 1450.00  ; 1#腔体机构在初始位
ORLD
AND 1455.02  ; 1#腔体机构自动/单次循环
OUT 1456.01  ; 1#腔体机构步进条件

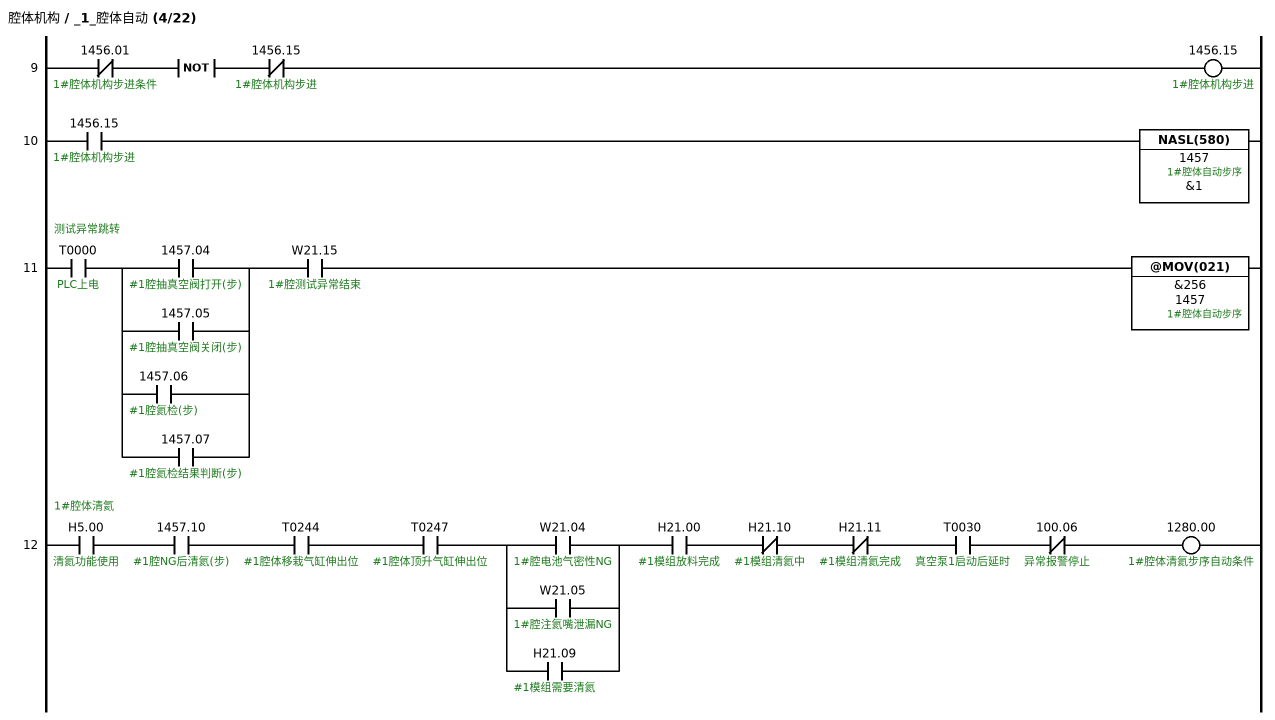
; rung 9
LDNOT 1456.01  ; 1#腔体机构步进条件
NOT(520)
ANDNOT 1456.15  ; 1#腔体机构步进
OUT 1456.15  ; 1#腔体机构步进
; rung 10
LD 1456.15  ; 1#腔体机构步进
NASL(580) 1457 &1  ; 1#腔体自动步序
; rung 11: 测试异常跳转
LD T0000  ; PLC上电
LD 1457.04  ; #1腔抽真空阀打开(步)
OR 1457.05  ; #1腔抽真空阀关闭(步)
OR 1457.06  ; #1腔氦检(步)
OR 1457.07  ; #1腔氦检结果判断(步)
ANDLD
AND W21.15  ; 1#腔测试异常结束
@MOV(021) &256 1457  ; 1#腔体自动步序
; rung 12: 1#腔体清氦
LD H5.00  ; 清氦功能使用
AND 1457.10  ; #1腔NG后清氦(步)
AND T0244  ; #1腔体移栽气缸伸出位
AND T0247  ; #1腔体顶升气缸伸出位
LD W21.04  ; 1#腔电池气密性NG
OR W21.05  ; 1#腔注氦嘴泄漏NG
OR H21.09  ; #1模组需要清氦
ANDLD
AND H21.00  ; #1模组放料完成
ANDNOT H21.10  ; #1模组清氦中
ANDNOT H21.11  ; #1模组清氦完成
AND T0030  ; 真空泵1启动后延时
ANDNOT 100.06  ; 异常报警停止
OUT 1280.00  ; 1#腔体清氦步序自动条件

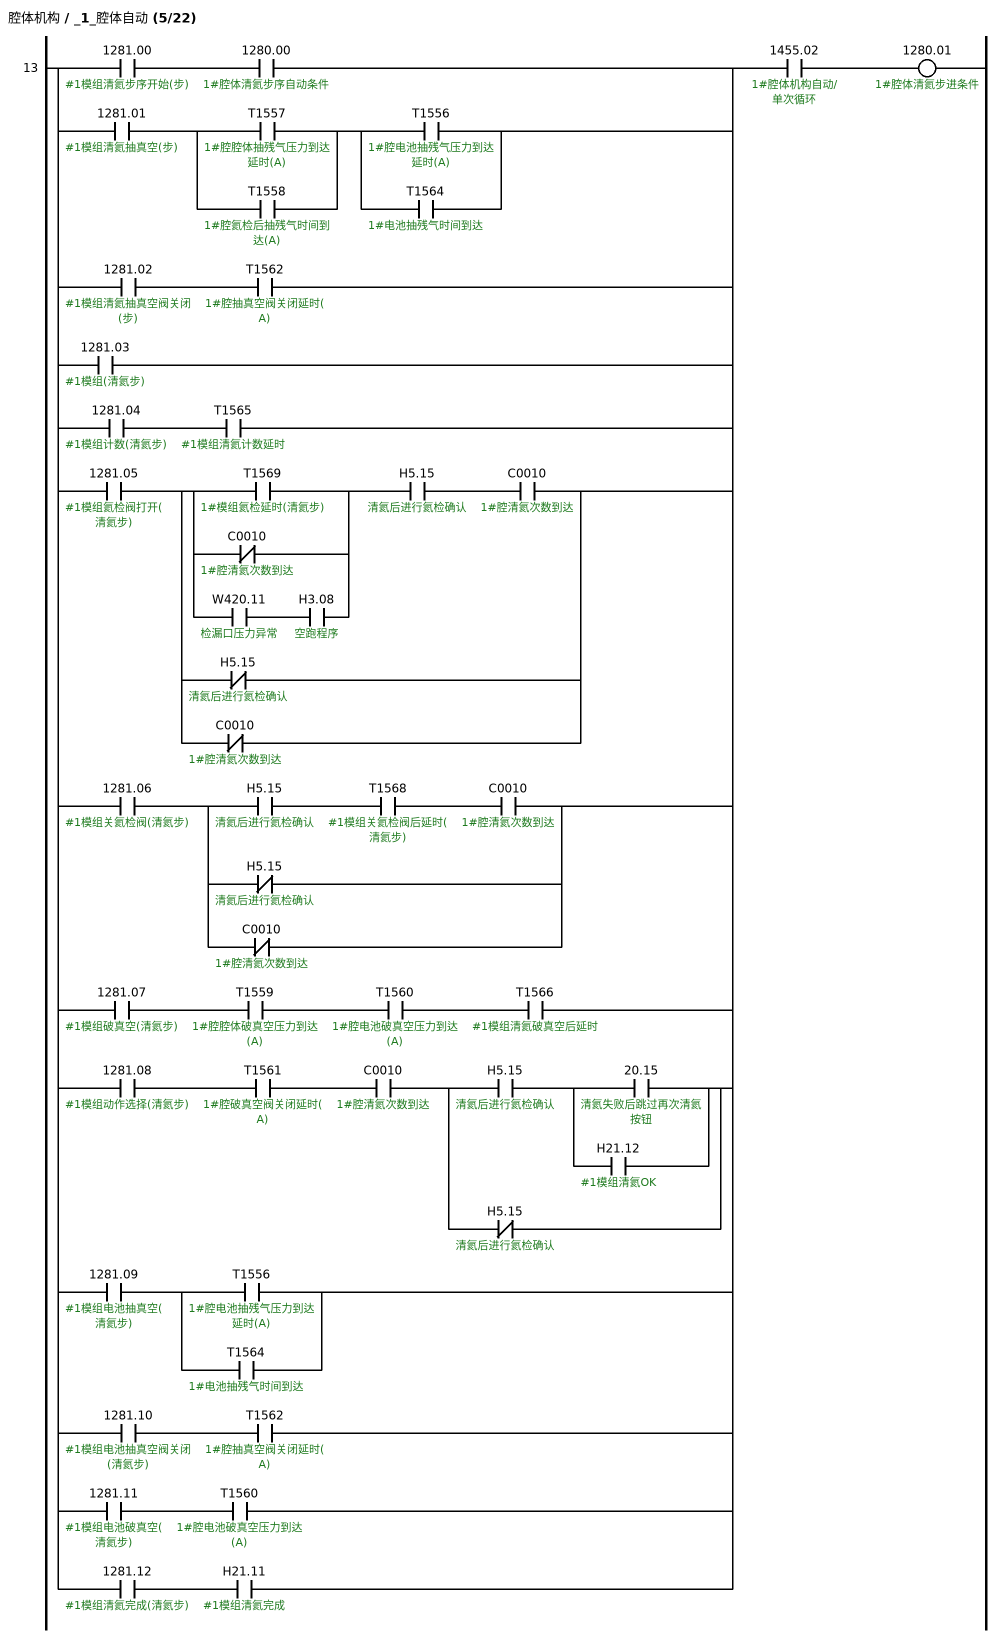
; rung 13
LD 1281.00  ; #1模组清氦步序开始(步)
AND 1280.00  ; 1#腔体清氦步序自动条件
LD 1281.01  ; #1模组清氦抽真空(步)
LD T1557  ; 1#腔腔体抽残气压力到达延时(A)
OR T1558  ; 1#腔氦检后抽残气时间到达(A)
ANDLD
LD T1556  ; 1#腔电池抽残气压力到达延时(A)
OR T1564  ; 1#电池抽残气时间到达
ANDLD
ORLD
LD 1281.02  ; #1模组清氦抽真空阀关闭(步)
AND T1562  ; 1#腔抽真空阀关闭延时(A)
ORLD
OR 1281.03  ; #1模组(清氦步)
LD 1281.04  ; #1模组计数(清氦步)
AND T1565  ; #1模组清氦计数延时
ORLD
LD 1281.05  ; #1模组氦检阀打开(清氦步)
LD T1569  ; 1#模组氦检延时(清氦步)
ORNOT C0010  ; 1#腔清氦次数到达
LD W420.11  ; 检漏口压力异常
AND H3.08  ; 空跑程序
ORLD
AND H5.15  ; 清氦后进行氦检确认
AND C0010  ; 1#腔清氦次数到达
ORNOT H5.15  ; 清氦后进行氦检确认
ORNOT C0010  ; 1#腔清氦次数到达
ANDLD
ORLD
LD 1281.06  ; #1模组关氦检阀(清氦步)
LD H5.15  ; 清氦后进行氦检确认
AND T1568  ; #1模组关氦检阀后延时(清氦步)
AND C0010  ; 1#腔清氦次数到达
ORNOT H5.15  ; 清氦后进行氦检确认
ORNOT C0010  ; 1#腔清氦次数到达
ANDLD
ORLD
LD 1281.07  ; #1模组破真空(清氦步)
AND T1559  ; 1#腔腔体破真空压力到达(A)
AND T1560  ; 1#腔电池破真空压力到达(A)
AND T1566  ; #1模组清氦破真空后延时
ORLD
LD 1281.08  ; #1模组动作选择(清氦步)
AND T1561  ; 1#腔破真空阀关闭延时(A)
AND C0010  ; 1#腔清氦次数到达
LD H5.15  ; 清氦后进行氦检确认
LD 20.15  ; 清氦失败后跳过再次清氦按钮
OR H21.12  ; #1模组清氦OK
ANDLD
ORNOT H5.15  ; 清氦后进行氦检确认
ANDLD
ORLD
LD 1281.09  ; #1模组电池抽真空(清氦步)
LD T1556  ; 1#腔电池抽残气压力到达延时(A)
OR T1564  ; 1#电池抽残气时间到达
ANDLD
ORLD
LD 1281.10  ; #1模组电池抽真空阀关闭(清氦步)
AND T1562  ; 1#腔抽真空阀关闭延时(A)
ORLD
LD 1281.11  ; #1模组电池破真空(清氦步)
AND T1560  ; 1#腔电池破真空压力到达(A)
ORLD
LD 1281.12  ; #1模组清氦完成(清氦步)
AND H21.11  ; #1模组清氦完成
ORLD
AND 1455.02  ; 1#腔体机构自动/单次循环
OUT 1280.01  ; 1#腔体清氦步进条件

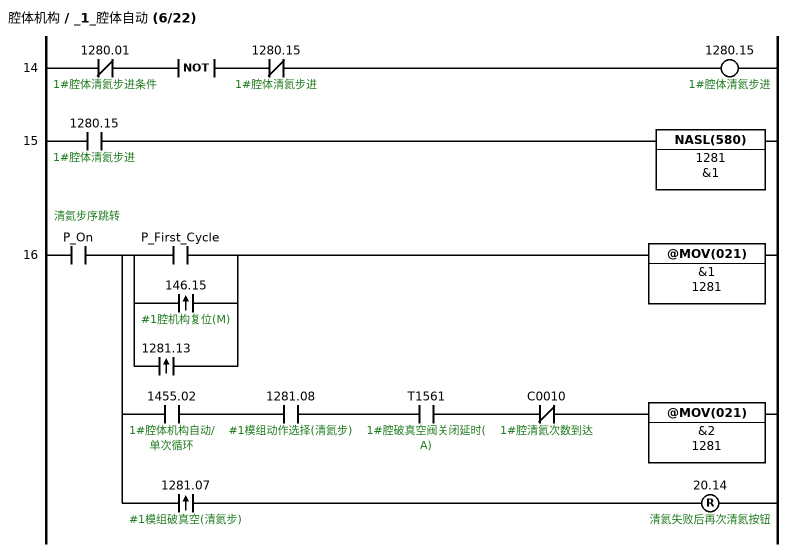
; rung 14
LDNOT 1280.01  ; 1#腔体清氦步进条件
NOT(520)
ANDNOT 1280.15  ; 1#腔体清氦步进
OUT 1280.15  ; 1#腔体清氦步进
; rung 15
LD 1280.15  ; 1#腔体清氦步进
NASL(580) 1281 &1
; rung 16: 清氦步序跳转
LD P_On
OUT TR0
LD P_First_Cycle
@OR 146.15  ; #1腔机构复位(M)
@OR 1281.13
ANDLD
@MOV(021) &1 1281
LD TR0
AND 1455.02  ; 1#腔体机构自动/单次循环
AND 1281.08  ; #1模组动作选择(清氦步)
AND T1561  ; 1#腔破真空阀关闭延时(A)
ANDNOT C0010  ; 1#腔清氦次数到达
@MOV(021) &2 1281
LD TR0
@AND 1281.07  ; #1模组破真空(清氦步)
RSET 20.14  ; 清氦失败后再次清氦按钮

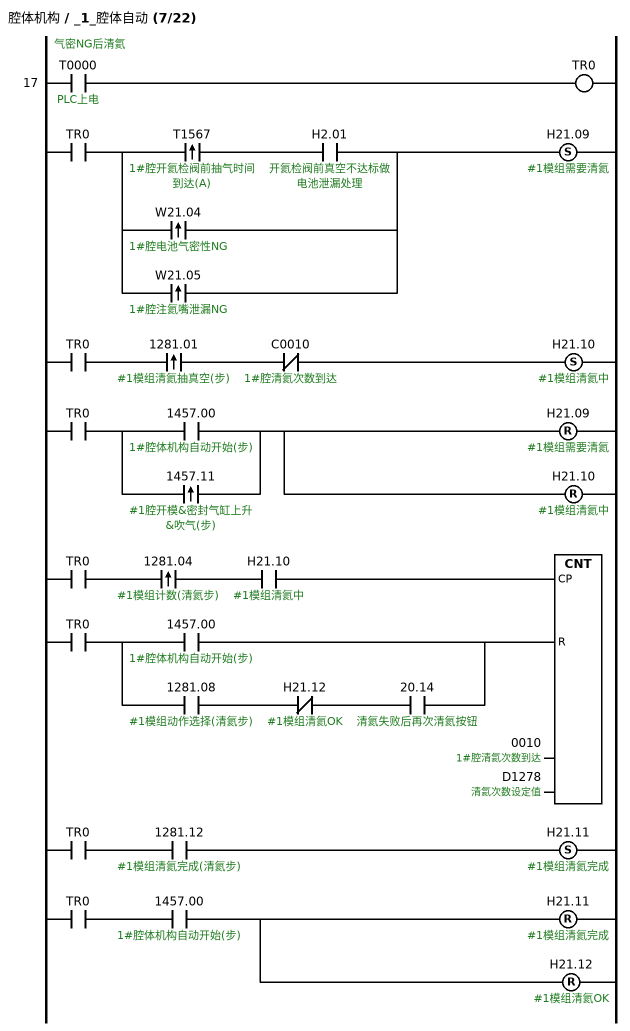
; rung 17: 气密NG后清氦
LD T0000  ; PLC上电
OUT TR0
@LD T1567  ; 1#腔开氦检阀前抽气时间到达(A)
AND H2.01  ; 开氦检阀前真空不达标做电池泄漏处理
@OR W21.04  ; 1#腔电池气密性NG
@OR W21.05  ; 1#腔注氦嘴泄漏NG
ANDLD
SET H21.09  ; #1模组需要清氦
LD TR0
@AND 1281.01  ; #1模组清氦抽真空(步)
ANDNOT C0010  ; 1#腔清氦次数到达
SET H21.10  ; #1模组清氦中
LD TR0
LD 1457.00  ; 1#腔体机构自动开始(步)
@OR 1457.11  ; #1腔开模&密封气缸上升&吹气(步)
ANDLD
RSET H21.09  ; #1模组需要清氦
RSET H21.10  ; #1模组清氦中
LD TR0
@AND 1281.04  ; #1模组计数(清氦步)
AND H21.10  ; #1模组清氦中
LD TR0
LD 1457.00  ; 1#腔体机构自动开始(步)
LD 1281.08  ; #1模组动作选择(清氦步)
ANDNOT H21.12  ; #1模组清氦OK
AND 20.14  ; 清氦失败后再次清氦按钮
ORLD
ANDLD
CNT 0010 D1278  ; 清氦次数设定值, 1#腔清氦次数到达
LD TR0
AND 1281.12  ; #1模组清氦完成(清氦步)
SET H21.11  ; #1模组清氦完成
LD TR0
AND 1457.00  ; 1#腔体机构自动开始(步)
RSET H21.11  ; #1模组清氦完成
RSET H21.12  ; #1模组清氦OK

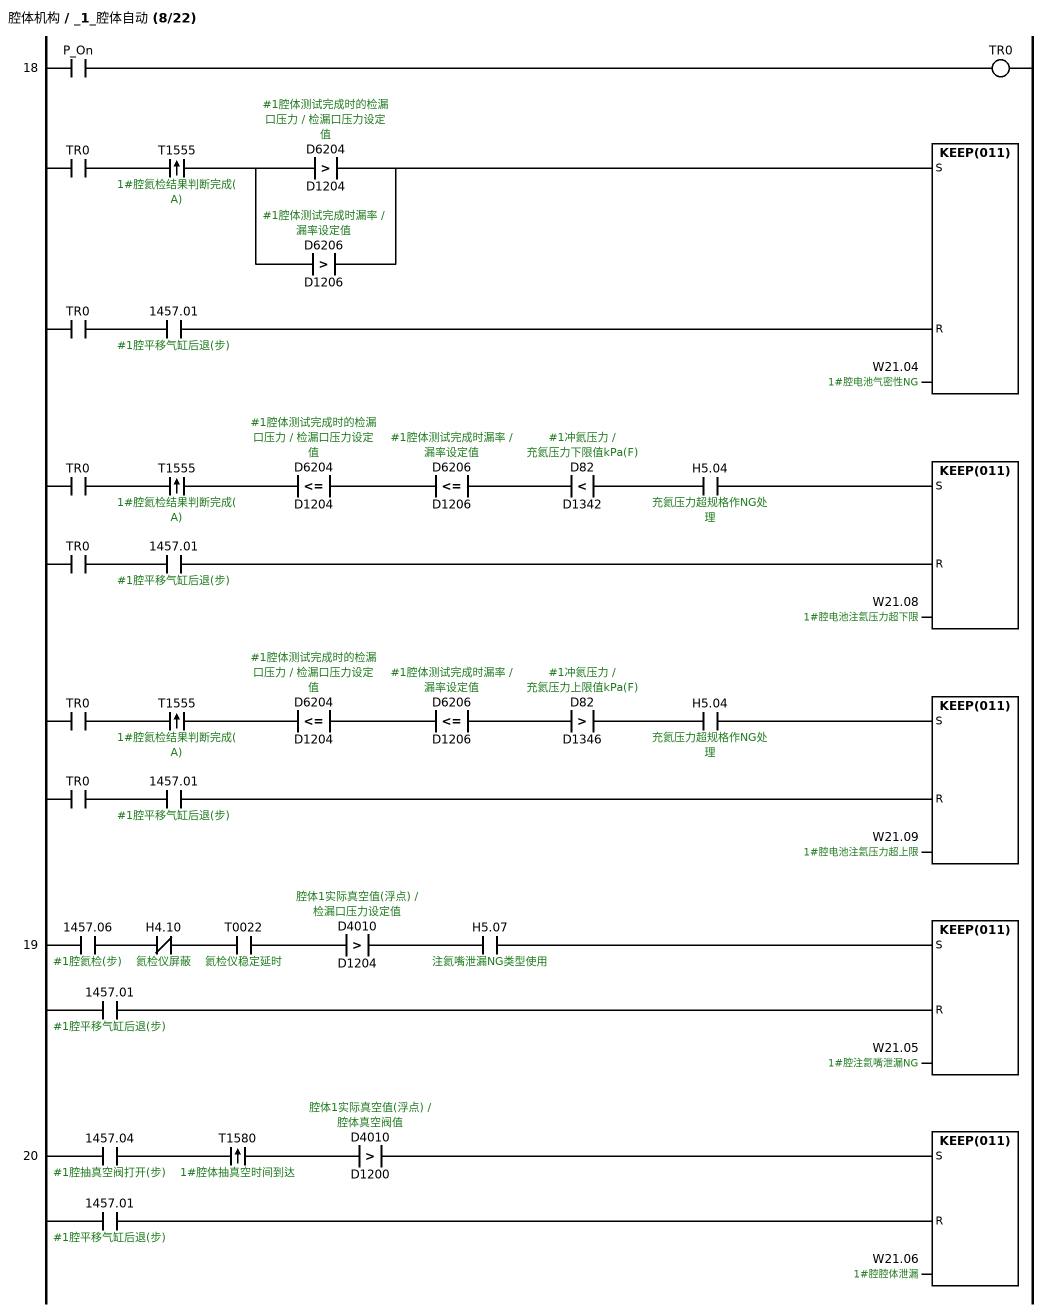
; rung 18
LD P_On
OUT TR0
@AND T1555  ; 1#腔氦检结果判断完成(A)
LD>F(333) D6204 D1204  ; #1腔体测试完成时的检漏口压力, 检漏口压力设定值
OR>F(333) D6206 D1206  ; #1腔体测试完成时漏率, 漏率设定值
ANDLD
LD TR0
AND 1457.01  ; #1腔平移气缸后退(步)
KEEP(011) W21.04  ; 1#腔电池气密性NG
LD TR0
@AND T1555  ; 1#腔氦检结果判断完成(A)
AND<=F(332) D6204 D1204  ; #1腔体测试完成时的检漏口压力, 检漏口压力设定值
AND<=F(332) D6206 D1206  ; #1腔体测试完成时漏率, 漏率设定值
AND<F(331) D82 D1342  ; #1冲氦压力, 充氦压力下限值kPa(F)
AND H5.04  ; 充氦压力超规格作NG处理
LD TR0
AND 1457.01  ; #1腔平移气缸后退(步)
KEEP(011) W21.08  ; 1#腔电池注氦压力超下限
LD TR0
@AND T1555  ; 1#腔氦检结果判断完成(A)
AND<=F(332) D6204 D1204  ; #1腔体测试完成时的检漏口压力, 检漏口压力设定值
AND<=F(332) D6206 D1206  ; #1腔体测试完成时漏率, 漏率设定值
AND>F(333) D82 D1346  ; #1冲氦压力, 充氦压力上限值kPa(F)
AND H5.04  ; 充氦压力超规格作NG处理
LD TR0
AND 1457.01  ; #1腔平移气缸后退(步)
KEEP(011) W21.09  ; 1#腔电池注氦压力超上限
; rung 19
LD 1457.06  ; #1腔氦检(步)
ANDNOT H4.10  ; 氦检仪屏蔽
AND T0022  ; 氦检仪稳定延时
AND>F(333) D4010 D1204  ; 腔体1实际真空值(浮点), 检漏口压力设定值
AND H5.07  ; 注氦嘴泄漏NG类型使用
LD 1457.01  ; #1腔平移气缸后退(步)
KEEP(011) W21.05  ; 1#腔注氦嘴泄漏NG
; rung 20
LD 1457.04  ; #1腔抽真空阀打开(步)
@AND T1580  ; 1#腔体抽真空时间到达
AND>F(333) D4010 D1200  ; 腔体1实际真空值(浮点), 腔体真空阀值
LD 1457.01  ; #1腔平移气缸后退(步)
KEEP(011) W21.06  ; 1#腔腔体泄漏

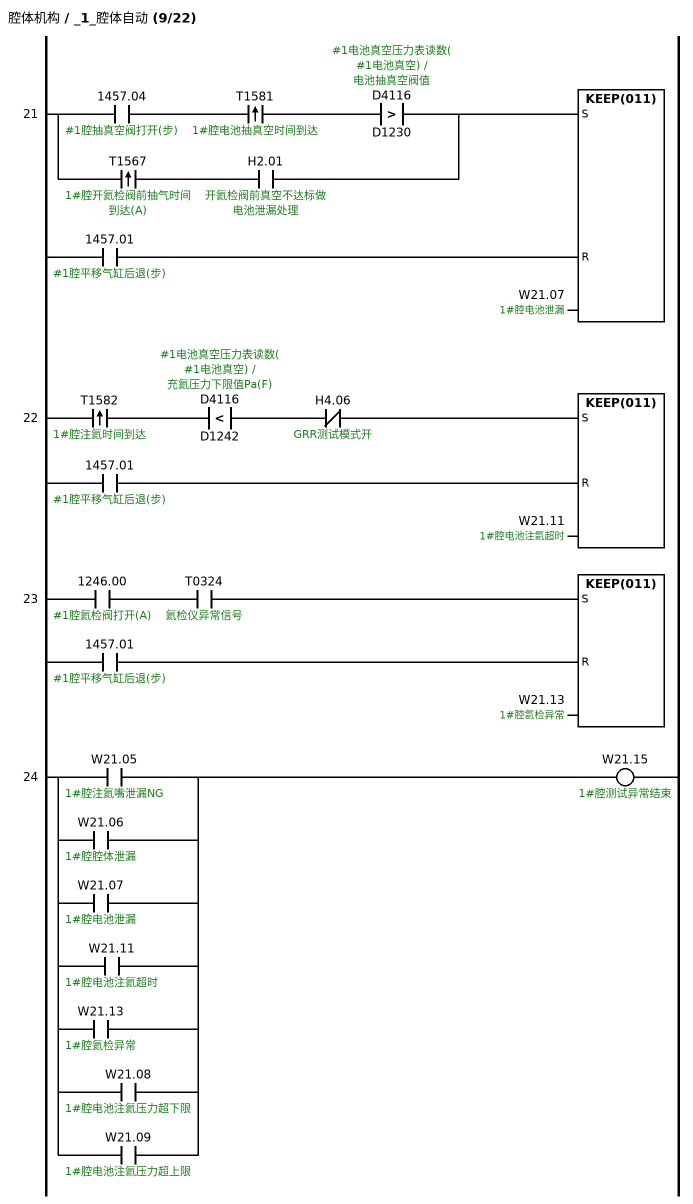
; rung 21
LD 1457.04  ; #1腔抽真空阀打开(步)
@AND T1581  ; 1#腔电池抽真空时间到达
AND>F(333) D4116 D1230  ; #1电池真空压力表读数(#1电池真空), 电池抽真空阀值
@LD T1567  ; 1#腔开氦检阀前抽气时间到达(A)
AND H2.01  ; 开氦检阀前真空不达标做电池泄漏处理
ORLD
LD 1457.01  ; #1腔平移气缸后退(步)
KEEP(011) W21.07  ; 1#腔电池泄漏
; rung 22
@LD T1582  ; 1#腔注氦时间到达
AND<F(331) D4116 D1242  ; #1电池真空压力表读数(#1电池真空), 充氦压力下限值Pa(F)
ANDNOT H4.06  ; GRR测试模式开
LD 1457.01  ; #1腔平移气缸后退(步)
KEEP(011) W21.11  ; 1#腔电池注氦超时
; rung 23
LD 1246.00  ; #1腔氦检阀打开(A)
AND T0324  ; 氦检仪异常信号
LD 1457.01  ; #1腔平移气缸后退(步)
KEEP(011) W21.13  ; 1#腔氦检异常
; rung 24
LD W21.05  ; 1#腔注氦嘴泄漏NG
OR W21.06  ; 1#腔腔体泄漏
OR W21.07  ; 1#腔电池泄漏
OR W21.11  ; 1#腔电池注氦超时
OR W21.13  ; 1#腔氦检异常
OR W21.08  ; 1#腔电池注氦压力超下限
OR W21.09  ; 1#腔电池注氦压力超上限
OUT W21.15  ; 1#腔测试异常结束

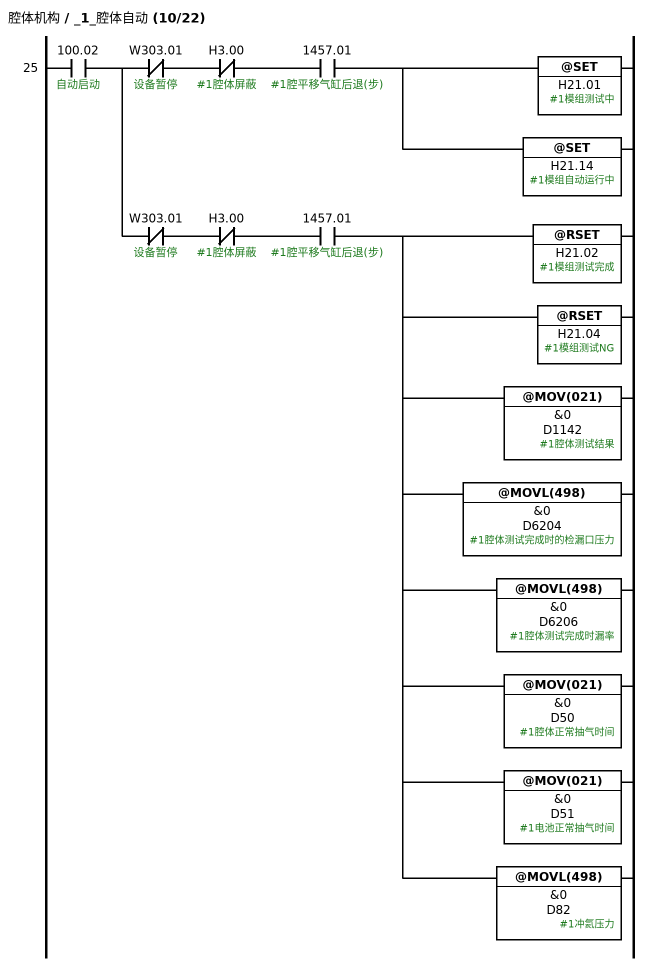
; rung 25
LD 100.02  ; 自动启动
OUT TR0
ANDNOT W303.01  ; 设备暂停
ANDNOT H3.00  ; #1腔体屏蔽
AND 1457.01  ; #1腔平移气缸后退(步)
@SET H21.01  ; #1模组测试中
@SET H21.14  ; #1模组自动运行中
LD TR0
ANDNOT W303.01  ; 设备暂停
ANDNOT H3.00  ; #1腔体屏蔽
AND 1457.01  ; #1腔平移气缸后退(步)
@RSET H21.02  ; #1模组测试完成
@RSET H21.04  ; #1模组测试NG
@MOV(021) &0 D1142  ; #1腔体测试结果
@MOVL(498) &0 D6204  ; #1腔体测试完成时的检漏口压力
@MOVL(498) &0 D6206  ; #1腔体测试完成时漏率
@MOV(021) &0 D50  ; #1腔体正常抽气时间
@MOV(021) &0 D51  ; #1电池正常抽气时间
@MOVL(498) &0 D82  ; #1冲氦压力

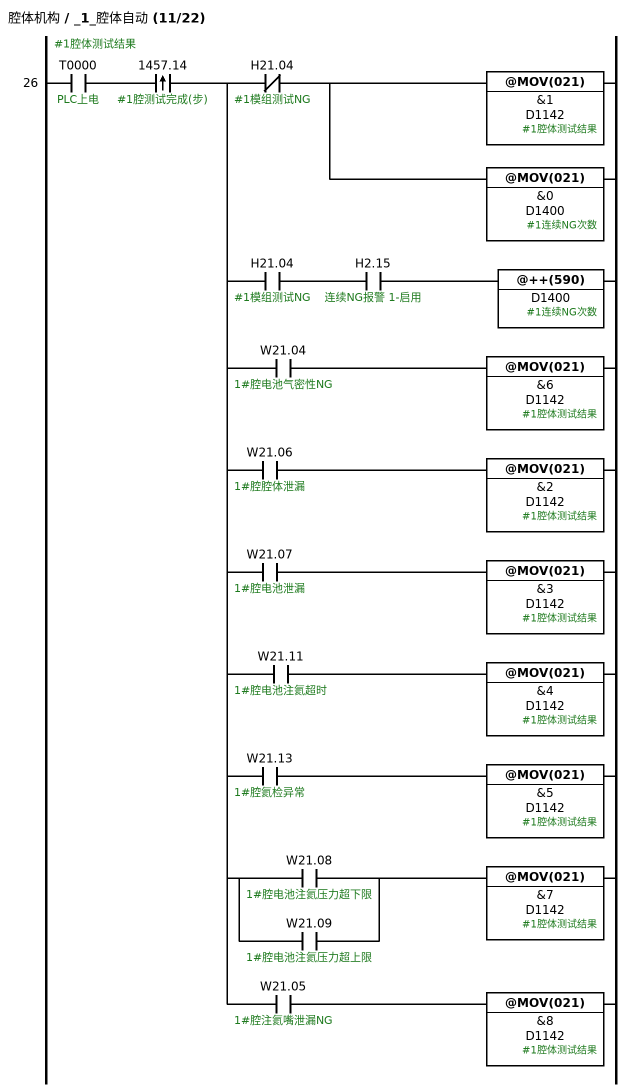
; rung 26: #1腔体测试结果
LD T0000  ; PLC上电
@AND 1457.14  ; #1腔测试完成(步)
OUT TR0
ANDNOT H21.04  ; #1模组测试NG
@MOV(021) &1 D1142  ; #1腔体测试结果
@MOV(021) &0 D1400  ; #1连续NG次数
LD TR0
AND H21.04  ; #1模组测试NG
AND H2.15  ; 连续NG报警 1-启用
@++(590) D1400  ; #1连续NG次数
LD TR0
AND W21.04  ; 1#腔电池气密性NG
@MOV(021) &6 D1142  ; #1腔体测试结果
LD TR0
AND W21.06  ; 1#腔腔体泄漏
@MOV(021) &2 D1142  ; #1腔体测试结果
LD TR0
AND W21.07  ; 1#腔电池泄漏
@MOV(021) &3 D1142  ; #1腔体测试结果
LD TR0
AND W21.11  ; 1#腔电池注氦超时
@MOV(021) &4 D1142  ; #1腔体测试结果
LD TR0
AND W21.13  ; 1#腔氦检异常
@MOV(021) &5 D1142  ; #1腔体测试结果
LD TR0
LD W21.08  ; 1#腔电池注氦压力超下限
OR W21.09  ; 1#腔电池注氦压力超上限
ANDLD
@MOV(021) &7 D1142  ; #1腔体测试结果
LD TR0
AND W21.05  ; 1#腔注氦嘴泄漏NG
@MOV(021) &8 D1142  ; #1腔体测试结果

